  MoveL 1304 to (49.51, 43.02, 7) mm, rotated rx 0 ry 90 rz 0 deg; joints [-9.498, 3.635, 52.807, 168.647, 56.961, -173.753]
  Set speed (120.0 mm/s)
  MoveL 1305 to (57.59, 48.33, 7) mm, rotated rx 0 ry 90 rz 0 deg; joints [-9.745, 4.388, 50.732, 168.176, 55.695, -173.271]
  Set speed (1000.0 mm/s)
  MoveL 1306 to (57.66, 48.4, 7) mm, rotated rx 0 ry 90 rz 0 deg; joints [-9.748, 4.395, 50.713, 168.17, 55.683, -173.265]
  Set speed (30.0 mm/s)
  Call Extruder(793.550)
  MoveL 1307 to (57.66, 50.87, 7) mm, rotated rx 0 ry 90 rz 0 deg; joints [-9.903, 4.432, 50.611, 167.975, 55.638, -173.145]
  Call Extruder(793.809)
  MoveL 1308 to (59.6, 50.88, 7) mm, rotated rx 0 ry 90 rz 0 deg; joints [-9.882, 4.602, 50.15, 167.959, 55.35, -173.085]
  Call Extruder(794.969)
  MoveL 1309 to (59.6, 59.6, 7) mm, rotated rx 0 ry 90 rz 0 deg; joints [-10.423, 4.74, 49.776, 167.271, 55.187, -172.651]
  Call Extruder(797.524)
  MoveL 1310 to (40.4, 59.6, 7) mm, rotated rx 0 ry 90 rz 0 deg; joints [-10.646, 3.144, 54.181, 167.412, 57.955, -173.243]
  Call Extruder(800.078)
  MoveL 1311 to (40.4, 40.4, 7) mm, rotated rx 0 ry 90 rz 0 deg; joints [-9.429, 2.881, 54.923, 168.897, 58.29, -174.111]
  Call Extruder(800.872)
  MoveL 1312 to (46.37, 40.4, 7) mm, rotated rx 0 ry 90 rz 0 deg; joints [-9.366, 3.347, 53.61, 168.868, 57.452, -173.957]
  Call Extruder(801.125)
  MoveL 1313 to (46.37, 42.3, 7) mm, rotated rx 0 ry 90 rz 0 deg; joints [-9.486, 3.372, 53.539, 168.721, 57.42, -173.871]
  Call Extruder(801.408)
  MoveL 1314 to (48.5, 42.29, 7) mm, rotated rx 0 ry 90 rz 0 deg; joints [-9.463, 3.543, 53.062, 168.71, 57.118, -173.814]
  Call Extruder(801.461)
  MoveL 1315 to (48.9, 42.29, 7) mm, rotated rx 0 ry 90 rz 0 deg; joints [-9.459, 3.575, 52.972, 168.707, 57.06, -173.803]
  Call Extruder(801.495)
  MoveL 1316 to (48.9, 41.89, 7) mm, rotated rx 0 ry 90 rz 0 deg; joints [-9.434, 3.57, 52.987, 168.738, 57.067, -173.821]
  Call Extruder(801.694)
  MoveL 1317 to (48.9, 40.4, 7) mm, rotated rx 0 ry 90 rz 0 deg; joints [-9.34, 3.55, 53.043, 168.854, 57.092, -173.89]
  Call Extruder(801.871)
  MoveL 1318 to (50.23, 40.4, 7) mm, rotated rx 0 ry 90 rz 0 deg; joints [-9.326, 3.658, 52.742, 168.846, 56.901, -173.855]
  Call Extruder(802.070)
  MoveL 1319 to (50.23, 41.9, 7) mm, rotated rx 0 ry 90 rz 0 deg; joints [-9.42, 3.678, 52.686, 168.73, 56.876, -173.785]
  Call Extruder(802.124)
  MoveL 1320 to (50.23, 42.3, 7) mm, rotated rx 0 ry 90 rz 0 deg; joints [-9.445, 3.683, 52.671, 168.699, 56.87, -173.767]
  Call Extruder(802.158)
  MoveL 1321 to (50.63, 42.3, 7) mm, rotated rx 0 ry 90 rz 0 deg; joints [-9.441, 3.716, 52.58, 168.697, 56.812, -173.756]
  Call Extruder(802.438)
  MoveL 1322 to (52.74, 42.3, 7) mm, rotated rx 0 ry 90 rz 0 deg; joints [-9.419, 3.89, 52.098, 168.683, 56.508, -173.698]
  Call Extruder(802.691)
  MoveL 1323 to (52.74, 40.4, 7) mm, rotated rx 0 ry 90 rz 0 deg; joints [-9.3, 3.865, 52.169, 168.831, 56.54, -173.787]
  Call Extruder(803.603)
  MoveL 1324 to (59.6, 40.4, 7) mm, rotated rx 0 ry 90 rz 0 deg; joints [-9.23, 4.447, 50.57, 168.782, 55.535, -173.596]
  Call Extruder(804.666)
  MoveL 1325 to (59.6, 48.39, 7) mm, rotated rx 0 ry 90 rz 0 deg; joints [-9.728, 4.564, 50.252, 168.154, 55.395, -173.207]
  Call Extruder(804.925)
  MoveL 1326 to (57.66, 48.4, 7) mm, rotated rx 0 ry 90 rz 0 deg; joints [-9.748, 4.395, 50.713, 168.17, 55.683, -173.265]
  Set speed (120.0 mm/s)
  MoveL 1327 to (57.66, 48.8, 7) mm, rotated rx 0 ry 90 rz 0 deg; joints [-9.773, 4.401, 50.697, 168.139, 55.676, -173.246]
  Set speed (1000.0 mm/s)
  MoveL 1328 to (57.56, 48.8, 7) mm, rotated rx 0 ry 90 rz 0 deg; joints [-9.774, 4.392, 50.72, 168.139, 55.691, -173.249]
  MoveL 1329 to (49.86, 42.5, 7) mm, rotated rx 0 ry 90 rz 0 deg; joints [-9.462, 3.656, 52.748, 168.685, 56.92, -173.767]
  MoveL 1330 to (49.57, 42.21, 7) mm, rotated rx 0 ry 90 rz 0 deg; joints [-9.447, 3.628, 52.825, 168.71, 56.967, -173.789]
  Set speed (30.0 mm/s)
  Call Extruder(804.972)
  MoveL 1331 to (49.57, 41.65, 7) mm, rotated rx 0 ry 90 rz 0 deg; joints [-9.411, 3.62, 52.846, 168.754, 56.976, -173.815]
  Call Extruder(805.055)
  MoveL 1332 to (49.4, 42.61, 7) mm, rotated rx 0 ry 90 rz 0 deg; joints [-9.474, 3.62, 52.848, 168.68, 56.984, -173.775]
  Set speed (120.0 mm/s)
  MoveL 1333 to (49.47, 42.86, 7) mm, rotated rx 0 ry 90 rz 0 deg; joints [-9.489, 3.629, 52.823, 168.66, 56.97, -173.762]
  Set speed (1000.0 mm/s)
  MoveL 1334 to (49.27, 43.01, 7) mm, rotated rx 0 ry 90 rz 0 deg; joints [-9.501, 3.615, 52.862, 168.649, 56.996, -173.76]
  MoveL 1335 to (49.27, 43.01, 7.4) mm, rotated rx 0 ry 90 rz 0 deg; joints [-9.501, 3.572, 52.909, 168.65, 56.999, -173.761]
  Set speed (60.0 mm/s)
  Call Extruder(805.506)
  MoveL 1336 to (45.88, 43.01, 7.4) mm, rotated rx 0 ry 90 rz 0 deg; joints [-9.537, 3.299, 53.669, 168.669, 57.482, -173.852]
  Call Extruder(805.533)
  MoveL 1337 to (45.88, 42.81, 7.4) mm, rotated rx 0 ry 90 rz 0 deg; joints [-9.524, 3.296, 53.677, 168.685, 57.486, -173.861]
  Call Extruder(806.428)
  MoveL 1338 to (41.12, 47.56, 7.4) mm, rotated rx 0 ry 90 rz 0 deg; joints [-9.876, 2.988, 54.547, 168.341, 58.073, -173.772]
  Call Extruder(807.286)
  MoveL 1339 to (41.12, 41.12, 7.4) mm, rotated rx 0 ry 90 rz 0 deg; joints [-9.467, 2.903, 54.786, 168.839, 58.181, -174.061]
  Call Extruder(810.627)
  MoveL 1340 to (58.88, 58.88, 7.4) mm, rotated rx 0 ry 90 rz 0 deg; joints [-10.386, 4.621, 50.029, 167.335, 55.313, -172.712]
  Call Extruder(810.627)
  MoveL 1341 to (58.88, 58.88, 7.4) mm, rotated rx 0 ry 90 rz 0 deg; joints [-10.386, 4.621, 50.029, 167.335, 55.313, -172.712]
  Call Extruder(811.485)
  MoveL 1342 to (58.88, 52.43, 7.4) mm, rotated rx 0 ry 90 rz 0 deg; joints [-9.986, 4.519, 50.306, 167.843, 55.434, -173.032]
  Call Extruder(812.698)
  MoveL 1343 to (52.43, 58.88, 7.4) mm, rotated rx 0 ry 90 rz 0 deg; joints [-10.46, 4.064, 51.546, 167.39, 56.26, -172.917]
  Call Extruder(813.345)
  MoveL 1344 to (47.57, 58.88, 7.4) mm, rotated rx 0 ry 90 rz 0 deg; joints [-10.516, 3.661, 52.661, 167.425, 56.961, -173.066]
  Call Extruder(814.558)
  MoveL 1345 to (41.12, 52.43, 7.4) mm, rotated rx 0 ry 90 rz 0 deg; joints [-10.184, 3.054, 54.358, 167.964, 57.988, -173.552]
  Call Extruder(815.416)
  MoveL 1346 to (41.12, 58.88, 7.4) mm, rotated rx 0 ry 90 rz 0 deg; joints [-10.592, 3.146, 54.099, 167.464, 57.871, -173.256]
  Call Extruder(815.416)
  MoveL 1347 to (41.12, 58.88, 7.4) mm, rotated rx 0 ry 90 rz 0 deg; joints [-10.592, 3.146, 54.099, 167.464, 57.871, -173.256]
  Call Extruder(818.758)
  MoveL 1348 to (58.88, 41.12, 7.4) mm, rotated rx 0 ry 90 rz 0 deg; joints [-9.282, 4.351, 50.761, 168.732, 55.634, -173.583]
  Call Extruder(819.615)
  MoveL 1349 to (58.88, 47.56, 7.4) mm, rotated rx 0 ry 90 rz 0 deg; joints [-9.684, 4.445, 50.506, 168.226, 55.522, -173.27]
  Call Extruder(820.682)
  MoveL 1350 to (53.21, 41.89, 7.4) mm, rotated rx 0 ry 90 rz 0 deg; joints [-9.389, 3.88, 52.054, 168.712, 56.451, -173.705]
  MoveL 1351 to (53.07, 41.75, 7.4) mm, rotated rx 0 ry 90 rz 0 deg; joints [-9.382, 3.866, 52.092, 168.724, 56.474, -173.716]
  Set speed (120.0 mm/s)
  MoveL 1352 to (49.27, 43.02, 7.4) mm, rotated rx 0 ry 90 rz 0 deg; joints [-9.501, 3.572, 52.909, 168.649, 56.999, -173.761]
  Set speed (60.0 mm/s)
  Call Extruder(821.206)
  MoveL 1353 to (53.21, 43.02, 7.4) mm, rotated rx 0 ry 90 rz 0 deg; joints [-9.459, 3.896, 52.011, 168.624, 56.432, -173.652]
  Call Extruder(821.458)
  MoveL 1354 to (53.21, 41.12, 7.4) mm, rotated rx 0 ry 90 rz 0 deg; joints [-9.34, 3.87, 52.082, 168.772, 56.464, -173.741]
  Call Extruder(822.213)
  MoveL 1355 to (58.88, 41.12, 7.4) mm, rotated rx 0 ry 90 rz 0 deg; joints [-9.282, 4.351, 50.761, 168.731, 55.634, -173.583]
  MoveL 1356 to (59.08, 41.12, 7.4) mm, rotated rx 0 ry 90 rz 0 deg; joints [-9.28, 4.369, 50.714, 168.73, 55.604, -173.577]
  Set speed (120.0 mm/s)
  MoveL 1357 to (49.27, 43.01, 7.4) mm, rotated rx 0 ry 90 rz 0 deg; joints [-9.501, 3.572, 52.909, 168.65, 56.999, -173.761]
  Set speed (60.0 mm/s)
  Call Extruder(822.213)
  MoveL 1358 to (49.27, 43.02, 7.4) mm, rotated rx 0 ry 90 rz 0 deg; joints [-9.501, 3.572, 52.909, 168.649, 56.999, -173.761]
  Set speed (120.0 mm/s)
  MoveL 1359 to (57.59, 48.32, 7.4) mm, rotated rx 0 ry 90 rz 0 deg; joints [-9.745, 4.344, 50.781, 168.177, 55.699, -173.272]
  Set speed (1000.0 mm/s)
  MoveL 1360 to (57.66, 48.39, 7.4) mm, rotated rx 0 ry 90 rz 0 deg; joints [-9.748, 4.351, 50.761, 168.171, 55.687, -173.267]
  Set speed (30.0 mm/s)
  Call Extruder(822.543)
  MoveL 1361 to (57.66, 50.87, 7.4) mm, rotated rx 0 ry 90 rz 0 deg; joints [-9.903, 4.388, 50.66, 167.976, 55.643, -173.146]
  Call Extruder(822.801)
  MoveL 1362 to (59.6, 50.87, 7.4) mm, rotated rx 0 ry 90 rz 0 deg; joints [-9.882, 4.558, 50.199, 167.96, 55.355, -173.086]
  Call Extruder(823.962)
  MoveL 1363 to (59.6, 59.6, 7.4) mm, rotated rx 0 ry 90 rz 0 deg; joints [-10.423, 4.696, 49.825, 167.271, 55.192, -172.653]
  Call Extruder(826.517)
  MoveL 1364 to (40.4, 59.6, 7.4) mm, rotated rx 0 ry 90 rz 0 deg; joints [-10.646, 3.101, 54.227, 167.412, 57.958, -173.244]
  Call Extruder(829.071)
  MoveL 1365 to (40.4, 40.4, 7.4) mm, rotated rx 0 ry 90 rz 0 deg; joints [-9.429, 2.839, 54.968, 168.898, 58.293, -174.112]
  Call Extruder(829.895)
  MoveL 1366 to (46.59, 40.4, 7.4) mm, rotated rx 0 ry 90 rz 0 deg; joints [-9.364, 3.322, 53.607, 168.868, 57.424, -173.952]
  Call Extruder(830.147)
  MoveL 1367 to (46.6, 42.29, 7.4) mm, rotated rx 0 ry 90 rz 0 deg; joints [-9.483, 3.347, 53.536, 168.721, 57.392, -173.866]
  Call Extruder(830.432)
  MoveL 1368 to (48.74, 42.29, 7.4) mm, rotated rx 0 ry 90 rz 0 deg; joints [-9.461, 3.519, 53.056, 168.709, 57.087, -173.808]
  Call Extruder(830.485)
  MoveL 1369 to (49.14, 42.29, 7.4) mm, rotated rx 0 ry 90 rz 0 deg; joints [-9.457, 3.551, 52.965, 168.706, 57.03, -173.797]
  Call Extruder(830.520)
  MoveL 1370 to (49.14, 41.89, 7.4) mm, rotated rx 0 ry 90 rz 0 deg; joints [-9.431, 3.546, 52.98, 168.737, 57.037, -173.816]
  Call Extruder(830.719)
  MoveL 1371 to (49.14, 40.4, 7.4) mm, rotated rx 0 ry 90 rz 0 deg; joints [-9.337, 3.526, 53.036, 168.853, 57.062, -173.885]
  Call Extruder(830.832)
  MoveL 1372 to (49.99, 40.4, 7.4) mm, rotated rx 0 ry 90 rz 0 deg; joints [-9.328, 3.595, 52.844, 168.848, 56.94, -173.862]
  Call Extruder(831.031)
  MoveL 1373 to (49.99, 41.9, 7.4) mm, rotated rx 0 ry 90 rz 0 deg; joints [-9.423, 3.615, 52.788, 168.732, 56.915, -173.793]
  Call Extruder(831.084)
  MoveL 1374 to (49.99, 42.29, 7.4) mm, rotated rx 0 ry 90 rz 0 deg; joints [-9.448, 3.62, 52.773, 168.701, 56.908, -173.774]
  Call Extruder(831.118)
  MoveL 1375 to (50.39, 42.3, 7.4) mm, rotated rx 0 ry 90 rz 0 deg; joints [-9.444, 3.653, 52.682, 168.699, 56.851, -173.764]
  Call Extruder(831.398)
  MoveL 1376 to (52.49, 42.3, 7.4) mm, rotated rx 0 ry 90 rz 0 deg; joints [-9.422, 3.826, 52.204, 168.685, 56.549, -173.706]
  Call Extruder(831.650)
  MoveL 1377 to (52.49, 40.4, 7.4) mm, rotated rx 0 ry 90 rz 0 deg; joints [-9.303, 3.8, 52.274, 168.833, 56.58, -173.795]
  Call Extruder(832.596)
  MoveL 1378 to (59.6, 40.4, 7.4) mm, rotated rx 0 ry 90 rz 0 deg; joints [-9.23, 4.404, 50.618, 168.782, 55.539, -173.597]
  Call Extruder(833.659)
  MoveL 1379 to (59.6, 48.39, 7.4) mm, rotated rx 0 ry 90 rz 0 deg; joints [-9.727, 4.52, 50.301, 168.155, 55.4, -173.208]
  Call Extruder(833.917)
  MoveL 1380 to (57.66, 48.39, 7.4) mm, rotated rx 0 ry 90 rz 0 deg; joints [-9.748, 4.351, 50.761, 168.171, 55.687, -173.267]
  Set speed (120.0 mm/s)
  MoveL 1381 to (57.66, 48.79, 7.4) mm, rotated rx 0 ry 90 rz 0 deg; joints [-9.773, 4.357, 50.745, 168.14, 55.68, -173.247]
  Set speed (1000.0 mm/s)
  MoveL 1382 to (57.56, 48.79, 7.4) mm, rotated rx 0 ry 90 rz 0 deg; joints [-9.774, 4.349, 50.769, 168.14, 55.695, -173.25]
  MoveL 1383 to (49.61, 42.59, 7.4) mm, rotated rx 0 ry 90 rz 0 deg; joints [-9.47, 3.594, 52.847, 168.68, 56.957, -173.771]
  MoveL 1384 to (49.56, 42.64, 7.4) mm, rotated rx 0 ry 90 rz 0 deg; joints [-9.474, 3.59, 52.857, 168.677, 56.964, -173.77]
  Set speed (30.0 mm/s)
  Call Extruder(833.929)
  MoveL 1385 to (49.56, 42.08, 7.4) mm, rotated rx 0 ry 90 rz 0 deg; joints [-9.439, 3.583, 52.878, 168.721, 56.973, -173.796]
  Call Extruder(833.954)
  MoveL 1386 to (49.56, 40.95, 7.4) mm, rotated rx 0 ry 90 rz 0 deg; joints [-9.367, 3.568, 52.92, 168.808, 56.992, -173.848]
  Set speed (120.0 mm/s)
  MoveL 1387 to (49.94, 40.9, 7.4) mm, rotated rx 0 ry 90 rz 0 deg; joints [-9.36, 3.597, 52.837, 168.81, 56.939, -173.841]
  Set speed (1000.0 mm/s)
  MoveL 1388 to (49.89, 40.9, 7.4) mm, rotated rx 0 ry 90 rz 0 deg; joints [-9.361, 3.594, 52.848, 168.81, 56.946, -173.842]
  MoveL 1389 to (49.02, 43.01, 7.4) mm, rotated rx 0 ry 90 rz 0 deg; joints [-9.503, 3.552, 52.964, 168.651, 57.035, -173.767]
  MoveL 1390 to (49.02, 43.01, 7.8) mm, rotated rx 0 ry 90 rz 0 deg; joints [-9.503, 3.509, 53.011, 168.651, 57.038, -173.768]
  Set speed (60.0 mm/s)
  Call Extruder(834.343)
  MoveL 1391 to (46.1, 43.02, 7.8) mm, rotated rx 0 ry 90 rz 0 deg; joints [-9.534, 3.274, 53.666, 168.668, 57.454, -173.847]
  Call Extruder(834.400)
  MoveL 1392 to (46.1, 42.59, 7.8) mm, rotated rx 0 ry 90 rz 0 deg; joints [-9.507, 3.268, 53.682, 168.701, 57.461, -173.866]
  Call Extruder(835.337)
  MoveL 1393 to (41.12, 47.56, 7.8) mm, rotated rx 0 ry 90 rz 0 deg; joints [-9.876, 2.945, 54.592, 168.341, 58.076, -173.773]
  Call Extruder(836.194)
  MoveL 1394 to (41.12, 41.12, 7.8) mm, rotated rx 0 ry 90 rz 0 deg; joints [-9.467, 2.86, 54.832, 168.839, 58.184, -174.062]
  Call Extruder(839.536)
  MoveL 1395 to (58.88, 58.88, 7.8) mm, rotated rx 0 ry 90 rz 0 deg; joints [-10.386, 4.577, 50.078, 167.336, 55.318, -172.714]
  Call Extruder(839.536)
  MoveL 1396 to (58.88, 58.88, 7.8) mm, rotated rx 0 ry 90 rz 0 deg; joints [-10.386, 4.577, 50.078, 167.336, 55.318, -172.714]
  Call Extruder(840.394)
  MoveL 1397 to (58.88, 52.43, 7.8) mm, rotated rx 0 ry 90 rz 0 deg; joints [-9.986, 4.475, 50.354, 167.844, 55.439, -173.033]
  Call Extruder(841.606)
  MoveL 1398 to (52.43, 58.88, 7.8) mm, rotated rx 0 ry 90 rz 0 deg; joints [-10.46, 4.021, 51.594, 167.39, 56.264, -172.918]
  Call Extruder(842.254)
  MoveL 1399 to (47.56, 58.88, 7.8) mm, rotated rx 0 ry 90 rz 0 deg; joints [-10.516, 3.618, 52.708, 167.425, 56.964, -173.067]
  Call Extruder(843.467)
  MoveL 1400 to (41.12, 52.43, 7.8) mm, rotated rx 0 ry 90 rz 0 deg; joints [-10.184, 3.012, 54.404, 167.964, 57.991, -173.552]
  Call Extruder(844.324)
  MoveL 1401 to (41.12, 58.88, 7.8) mm, rotated rx 0 ry 90 rz 0 deg; joints [-10.592, 3.104, 54.145, 167.464, 57.874, -173.257]
  Call Extruder(844.325)
  MoveL 1402 to (41.12, 58.88, 7.8) mm, rotated rx 0 ry 90 rz 0 deg; joints [-10.592, 3.104, 54.145, 167.464, 57.874, -173.257]
  Call Extruder(847.666)
  MoveL 1403 to (58.88, 41.12, 7.8) mm, rotated rx 0 ry 90 rz 0 deg; joints [-9.282, 4.308, 50.81, 168.732, 55.639, -173.584]
  Call Extruder(848.524)
  MoveL 1404 to (58.88, 47.56, 7.8) mm, rotated rx 0 ry 90 rz 0 deg; joints [-9.684, 4.401, 50.555, 168.227, 55.527, -173.272]
  Call Extruder(849.638)
  MoveL 1405 to (52.96, 41.64, 7.8) mm, rotated rx 0 ry 90 rz 0 deg; joints [-9.376, 3.812, 52.168, 168.734, 56.496, -173.725]
  MoveL 1406 to (52.81, 41.5, 7.8) mm, rotated rx 0 ry 90 rz 0 deg; joints [-9.368, 3.799, 52.206, 168.746, 56.519, -173.735]
  Set speed (120.0 mm/s)
  MoveL 1407 to (49.02, 43.02, 7.8) mm, rotated rx 0 ry 90 rz 0 deg; joints [-9.503, 3.509, 53.011, 168.651, 57.038, -173.768]
  Set speed (60.0 mm/s)
  Call Extruder(850.161)
  MoveL 1408 to (52.95, 43.02, 7.8) mm, rotated rx 0 ry 90 rz 0 deg; joints [-9.462, 3.831, 52.116, 168.626, 56.473, -173.66]
  Call Extruder(850.414)
  MoveL 1409 to (52.96, 41.12, 7.8) mm, rotated rx 0 ry 90 rz 0 deg; joints [-9.343, 3.805, 52.188, 168.774, 56.504, -173.749]
  Call Extruder(851.202)
  MoveL 1410 to (58.88, 41.12, 7.8) mm, rotated rx 0 ry 90 rz 0 deg; joints [-9.282, 4.308, 50.809, 168.732, 55.638, -173.584]
  MoveL 1411 to (59.08, 41.12, 7.8) mm, rotated rx 0 ry 90 rz 0 deg; joints [-9.28, 4.325, 50.762, 168.731, 55.609, -173.578]
  Set speed (120.0 mm/s)
  MoveL 1412 to (49.02, 43.01, 7.8) mm, rotated rx 0 ry 90 rz 0 deg; joints [-9.503, 3.509, 53.011, 168.651, 57.038, -173.768]
  Set speed (60.0 mm/s)
  Call Extruder(851.202)
  MoveL 1413 to (49.02, 43.02, 7.8) mm, rotated rx 0 ry 90 rz 0 deg; joints [-9.503, 3.509, 53.011, 168.651, 57.038, -173.768]
  Set speed (120.0 mm/s)
  MoveL 1414 to (49.74, 42.29, 7.8) mm, rotated rx 0 ry 90 rz 0 deg; joints [-9.45, 3.557, 52.875, 168.703, 56.947, -173.782]
  Set speed (30.0 mm/s)
  Call Extruder(851.533)
  MoveL 1415 to (52.24, 42.3, 7.8) mm, rotated rx 0 ry 90 rz 0 deg; joints [-9.424, 3.762, 52.309, 168.687, 56.589, -173.714]
  Call Extruder(851.785)
  MoveL 1416 to (52.24, 40.4, 7.8) mm, rotated rx 0 ry 90 rz 0 deg; joints [-9.305, 3.736, 52.379, 168.835, 56.62, -173.803]
  Call Extruder(852.765)
  MoveL 1417 to (59.6, 40.4, 7.8) mm, rotated rx 0 ry 90 rz 0 deg; joints [-9.23, 4.36, 50.667, 168.783, 55.544, -173.598]
  Call Extruder(853.827)
  MoveL 1418 to (59.6, 48.39, 7.8) mm, rotated rx 0 ry 90 rz 0 deg; joints [-9.727, 4.476, 50.35, 168.156, 55.405, -173.21]
  Call Extruder(854.032)
  MoveL 1419 to (58.06, 48.39, 7.8) mm, rotated rx 0 ry 90 rz 0 deg; joints [-9.744, 4.342, 50.715, 168.169, 55.633, -173.256]
  Call Extruder(854.085)
  MoveL 1420 to (57.66, 48.39, 7.8) mm, rotated rx 0 ry 90 rz 0 deg; joints [-9.748, 4.308, 50.81, 168.172, 55.692, -173.268]
  Call Extruder(854.120)
  MoveL 1421 to (57.66, 48.79, 7.8) mm, rotated rx 0 ry 90 rz 0 deg; joints [-9.773, 4.314, 50.793, 168.141, 55.685, -173.249]
  Call Extruder(854.396)
  MoveL 1422 to (57.66, 50.87, 7.8) mm, rotated rx 0 ry 90 rz 0 deg; joints [-9.902, 4.345, 50.708, 167.977, 55.647, -173.147]
  Call Extruder(854.654)
  MoveL 1423 to (59.6, 50.87, 7.8) mm, rotated rx 0 ry 90 rz 0 deg; joints [-9.881, 4.514, 50.248, 167.961, 55.36, -173.088]
  Call Extruder(855.816)
  MoveL 1424 to (59.6, 59.6, 7.8) mm, rotated rx 0 ry 90 rz 0 deg; joints [-10.423, 4.652, 49.874, 167.272, 55.197, -172.654]
  Call Extruder(858.370)
  MoveL 1425 to (40.4, 59.6, 7.8) mm, rotated rx 0 ry 90 rz 0 deg; joints [-10.646, 3.058, 54.273, 167.412, 57.961, -173.244]
  Call Extruder(860.925)
  MoveL 1426 to (40.4, 40.4, 7.8) mm, rotated rx 0 ry 90 rz 0 deg; joints [-9.429, 2.796, 55.014, 168.898, 58.296, -174.112]
  Call Extruder(861.778)
  MoveL 1427 to (46.82, 40.4, 7.8) mm, rotated rx 0 ry 90 rz 0 deg; joints [-9.361, 3.297, 53.603, 168.867, 57.396, -173.947]
  Call Extruder(862.030)
  MoveL 1428 to (46.82, 42.3, 7.8) mm, rotated rx 0 ry 90 rz 0 deg; joints [-9.481, 3.322, 53.533, 168.72, 57.364, -173.86]
  Call Extruder(862.371)
  MoveL 1429 to (49.37, 42.29, 7.8) mm, rotated rx 0 ry 90 rz 0 deg; joints [-9.454, 3.527, 52.959, 168.705, 57, -173.792]
  Call Extruder(862.474)
  MoveL 1430 to (49.37, 41.52, 7.8) mm, rotated rx 0 ry 90 rz 0 deg; joints [-9.405, 3.517, 52.988, 168.766, 57.013, -173.828]
  Call Extruder(862.623)
  MoveL 1431 to (49.37, 40.4, 7.8) mm, rotated rx 0 ry 90 rz 0 deg; joints [-9.335, 3.502, 53.029, 168.852, 57.032, -173.879]
  Call Extruder(862.672)
  MoveL 1432 to (49.75, 40.4, 7.8) mm, rotated rx 0 ry 90 rz 0 deg; joints [-9.331, 3.532, 52.945, 168.85, 56.978, -173.87]
  Call Extruder(862.741)
  MoveL 1433 to (49.75, 41.52, 7.8) mm, rotated rx 0 ry 90 rz 0 deg; joints [-9.401, 3.547, 52.904, 168.764, 56.96, -173.818]
  Call Extruder(862.789)
  MoveL 1434 to (49.74, 42.29, 7.8) mm, rotated rx 0 ry 90 rz 0 deg; joints [-9.45, 3.557, 52.875, 168.703, 56.947, -173.782]
  Set speed (120.0 mm/s)
  MoveL 1435 to (50.14, 42.29, 7.8) mm, rotated rx 0 ry 90 rz 0 deg; joints [-9.446, 3.59, 52.785, 168.701, 56.89, -173.771]
  Set speed (1000.0 mm/s)
  MoveL 1436 to (50.14, 43.1, 7.8) mm, rotated rx 0 ry 90 rz 0 deg; joints [-9.496, 3.601, 52.754, 168.638, 56.876, -173.734]
  MoveL 1437 to (52.26, 42.32, 7.8) mm, rotated rx 0 ry 90 rz 0 deg; joints [-9.426, 3.764, 52.301, 168.685, 56.585, -173.712]
  MoveL 1438 to (52.7, 41.39, 7.8) mm, rotated rx 0 ry 90 rz 0 deg; joints [-9.363, 3.788, 52.236, 168.755, 56.537, -173.744]
  MoveL 1439 to (52.7, 41.39, 8.2) mm, rotated rx 0 ry 90 rz 0 deg; joints [-9.363, 3.745, 52.283, 168.755, 56.541, -173.745]
  Set speed (60.0 mm/s)
  Call Extruder(863.951)
  MoveL 1440 to (58.88, 47.57, 8.2) mm, rotated rx 0 ry 90 rz 0 deg; joints [-9.684, 4.357, 50.603, 168.227, 55.531, -173.273]
  Call Extruder(864.809)
  MoveL 1441 to (58.88, 41.12, 8.2) mm, rotated rx 0 ry 90 rz 0 deg; joints [-9.282, 4.264, 50.858, 168.733, 55.643, -173.585]
  Call Extruder(868.150)
  MoveL 1442 to (41.12, 58.88, 8.2) mm, rotated rx 0 ry 90 rz 0 deg; joints [-10.592, 3.061, 54.191, 167.465, 57.877, -173.258]
  Call Extruder(868.151)
  MoveL 1443 to (41.12, 58.88, 8.2) mm, rotated rx 0 ry 90 rz 0 deg; joints [-10.592, 3.061, 54.19, 167.465, 57.877, -173.257]
  Call Extruder(869.008)
  MoveL 1444 to (41.12, 52.43, 8.2) mm, rotated rx 0 ry 90 rz 0 deg; joints [-10.184, 2.969, 54.45, 167.965, 57.994, -173.553]
  Call Extruder(870.221)
  MoveL 1445 to (47.57, 58.88, 8.2) mm, rotated rx 0 ry 90 rz 0 deg; joints [-10.516, 3.575, 52.755, 167.426, 56.968, -173.068]
  Call Extruder(870.869)
  MoveL 1446 to (52.43, 58.88, 8.2) mm, rotated rx 0 ry 90 rz 0 deg; joints [-10.46, 3.978, 51.642, 167.391, 56.268, -172.919]
  Call Extruder(872.082)
  MoveL 1447 to (58.88, 52.43, 8.2) mm, rotated rx 0 ry 90 rz 0 deg; joints [-9.986, 4.431, 50.403, 167.844, 55.443, -173.034]
  Call Extruder(872.939)
  MoveL 1448 to (58.88, 58.88, 8.2) mm, rotated rx 0 ry 90 rz 0 deg; joints [-10.386, 4.533, 50.127, 167.336, 55.323, -172.715]
  Call Extruder(872.940)
  MoveL 1449 to (58.88, 58.88, 8.2) mm, rotated rx 0 ry 90 rz 0 deg; joints [-10.386, 4.533, 50.127, 167.337, 55.323, -172.715]
  Call Extruder(876.281)
  MoveL 1450 to (41.12, 41.12, 8.2) mm, rotated rx 0 ry 90 rz 0 deg; joints [-9.467, 2.818, 54.877, 168.84, 58.187, -174.063]
  Call Extruder(877.139)
  MoveL 1451 to (41.12, 47.56, 8.2) mm, rotated rx 0 ry 90 rz 0 deg; joints [-9.876, 2.902, 54.638, 168.342, 58.079, -173.774]
  Call Extruder(878.117)
  MoveL 1452 to (46.32, 42.37, 8.2) mm, rotated rx 0 ry 90 rz 0 deg; joints [-9.491, 3.24, 53.687, 168.718, 57.437, -173.871]
  Call Extruder(878.203)
  MoveL 1453 to (46.32, 43.02, 8.2) mm, rotated rx 0 ry 90 rz 0 deg; joints [-9.532, 3.249, 53.663, 168.667, 57.426, -173.841]
  Call Extruder(879.052)
  MoveL 1454 to (52.7, 43.02, 8.2) mm, rotated rx 0 ry 90 rz 0 deg; joints [-9.465, 3.767, 52.222, 168.629, 56.513, -173.668]
  Call Extruder(879.304)
  MoveL 1455 to (52.7, 41.12, 8.2) mm, rotated rx 0 ry 90 rz 0 deg; joints [-9.346, 3.741, 52.293, 168.776, 56.545, -173.757]
  Call Extruder(880.126)
  MoveL 1456 to (58.88, 41.12, 8.2) mm, rotated rx 0 ry 90 rz 0 deg; joints [-9.282, 4.264, 50.858, 168.733, 55.643, -173.585]
  MoveL 1457 to (59.08, 41.12, 8.2) mm, rotated rx 0 ry 90 rz 0 deg; joints [-9.28, 4.281, 50.81, 168.731, 55.613, -173.579]
  Set speed (120.0 mm/s)
  MoveL 1458 to (57.59, 48.31, 8.2) mm, rotated rx 0 ry 90 rz 0 deg; joints [-9.744, 4.257, 50.877, 168.179, 55.708, -173.275]
  Set speed (1000.0 mm/s)
  MoveL 1459 to (57.66, 48.38, 8.2) mm, rotated rx 0 ry 90 rz 0 deg; joints [-9.748, 4.264, 50.858, 168.173, 55.696, -173.269]
  Set speed (30.0 mm/s)
  Call Extruder(880.353)
  MoveL 1460 to (57.66, 50.09, 8.2) mm, rotated rx 0 ry 90 rz 0 deg; joints [-9.854, 4.289, 50.789, 168.039, 55.666, -173.186]
  Call Extruder(880.456)
  MoveL 1461 to (57.66, 50.86, 8.2) mm, rotated rx 0 ry 90 rz 0 deg; joints [-9.902, 4.301, 50.756, 167.978, 55.652, -173.149]
  Call Extruder(880.714)
  MoveL 1462 to (59.6, 50.86, 8.2) mm, rotated rx 0 ry 90 rz 0 deg; joints [-9.881, 4.47, 50.297, 167.962, 55.365, -173.089]
  Call Extruder(881.876)
  MoveL 1463 to (59.6, 59.6, 8.2) mm, rotated rx 0 ry 90 rz 0 deg; joints [-10.423, 4.608, 49.923, 167.273, 55.202, -172.655]
  Call Extruder(884.430)
  MoveL 1464 to (40.4, 59.6, 8.2) mm, rotated rx 0 ry 90 rz 0 deg; joints [-10.646, 3.015, 54.319, 167.413, 57.964, -173.245]
  Call Extruder(886.985)
  MoveL 1465 to (40.4, 40.4, 8.2) mm, rotated rx 0 ry 90 rz 0 deg; joints [-9.429, 2.754, 55.059, 168.898, 58.299, -174.113]
  Call Extruder(887.868)
  MoveL 1466 to (47.04, 40.4, 8.2) mm, rotated rx 0 ry 90 rz 0 deg; joints [-9.359, 3.271, 53.6, 168.866, 57.368, -173.942]
  Call Extruder(888.120)
  MoveL 1467 to (47.04, 42.3, 8.2) mm, rotated rx 0 ry 90 rz 0 deg; joints [-9.479, 3.297, 53.529, 168.719, 57.336, -173.855]
  Call Extruder(888.778)
  MoveL 1468 to (51.98, 42.3, 8.2) mm, rotated rx 0 ry 90 rz 0 deg; joints [-9.427, 3.698, 52.413, 168.689, 56.629, -173.722]
  Call Extruder(889.030)
  MoveL 1469 to (51.99, 40.4, 8.2) mm, rotated rx 0 ry 90 rz 0 deg; joints [-9.308, 3.672, 52.484, 168.837, 56.661, -173.81]
  Call Extruder(890.043)
  MoveL 1470 to (59.6, 40.4, 8.2) mm, rotated rx 0 ry 90 rz 0 deg; joints [-9.23, 4.316, 50.715, 168.784, 55.549, -173.599]
  Call Extruder(891.105)
  MoveL 1471 to (59.6, 48.38, 8.2) mm, rotated rx 0 ry 90 rz 0 deg; joints [-9.727, 4.433, 50.399, 168.157, 55.41, -173.211]
  Call Extruder(891.363)
  MoveL 1472 to (57.66, 48.38, 8.2) mm, rotated rx 0 ry 90 rz 0 deg; joints [-9.748, 4.264, 50.858, 168.173, 55.696, -173.269]
  Set speed (120.0 mm/s)
  MoveL 1473 to (57.66, 48.78, 8.2) mm, rotated rx 0 ry 90 rz 0 deg; joints [-9.773, 4.27, 50.842, 168.142, 55.689, -173.25]
  Set speed (1000.0 mm/s)
  MoveL 1474 to (56.86, 48.78, 8.2) mm, rotated rx 0 ry 90 rz 0 deg; joints [-9.781, 4.201, 51.03, 168.148, 55.807, -173.274]
  MoveL 1475 to (52.45, 41.14, 8.2) mm, rotated rx 0 ry 90 rz 0 deg; joints [-9.349, 3.72, 52.351, 168.777, 56.581, -173.763]
  MoveL 1476 to (52.45, 41.14, 8.6) mm, rotated rx 0 ry 90 rz 0 deg; joints [-9.349, 3.677, 52.398, 168.777, 56.585, -173.764]
  Set speed (60.0 mm/s)
  Call Extruder(892.573)
  MoveL 1477 to (58.88, 47.57, 8.6) mm, rotated rx 0 ry 90 rz 0 deg; joints [-9.684, 4.314, 50.652, 168.228, 55.536, -173.274]
  Call Extruder(893.430)
  MoveL 1478 to (58.88, 41.12, 8.6) mm, rotated rx 0 ry 90 rz 0 deg; joints [-9.282, 4.22, 50.906, 168.733, 55.647, -173.586]
  Call Extruder(896.772)
  MoveL 1479 to (41.12, 58.88, 8.6) mm, rotated rx 0 ry 90 rz 0 deg; joints [-10.592, 3.018, 54.236, 167.465, 57.88, -173.258]
  Call Extruder(896.772)
  MoveL 1480 to (41.12, 58.88, 8.6) mm, rotated rx 0 ry 90 rz 0 deg; joints [-10.592, 3.018, 54.236, 167.465, 57.88, -173.258]
  Call Extruder(897.630)
  MoveL 1481 to (41.12, 52.43, 8.6) mm, rotated rx 0 ry 90 rz 0 deg; joints [-10.184, 2.926, 54.495, 167.965, 57.997, -173.554]
  Call Extruder(898.842)
  MoveL 1482 to (47.57, 58.88, 8.6) mm, rotated rx 0 ry 90 rz 0 deg; joints [-10.516, 3.532, 52.801, 167.426, 56.972, -173.068]
  Call Extruder(899.490)
  MoveL 1483 to (52.43, 58.88, 8.6) mm, rotated rx 0 ry 90 rz 0 deg; joints [-10.46, 3.934, 51.689, 167.391, 56.272, -172.92]
  Call Extruder(900.703)
  MoveL 1484 to (58.88, 52.43, 8.6) mm, rotated rx 0 ry 90 rz 0 deg; joints [-9.986, 4.387, 50.451, 167.845, 55.448, -173.036]
  Call Extruder(901.561)
  MoveL 1485 to (58.88, 58.88, 8.6) mm, rotated rx 0 ry 90 rz 0 deg; joints [-10.386, 4.489, 50.175, 167.337, 55.327, -172.716]
  Call Extruder(901.561)
  MoveL 1486 to (58.88, 58.88, 8.6) mm, rotated rx 0 ry 90 rz 0 deg; joints [-10.386, 4.489, 50.176, 167.337, 55.327, -172.716]
  Call Extruder(904.902)
  MoveL 1487 to (41.12, 41.12, 8.6) mm, rotated rx 0 ry 90 rz 0 deg; joints [-9.467, 2.775, 54.922, 168.84, 58.19, -174.063]
  Call Extruder(905.760)
  MoveL 1488 to (41.12, 47.56, 8.6) mm, rotated rx 0 ry 90 rz 0 deg; joints [-9.876, 2.86, 54.683, 168.342, 58.081, -173.774]
  Call Extruder(906.780)
  MoveL 1489 to (46.54, 42.14, 8.6) mm, rotated rx 0 ry 90 rz 0 deg; joints [-9.474, 3.212, 53.692, 168.734, 57.412, -173.876]
  Call Extruder(906.896)
  MoveL 1490 to (46.54, 43.02, 8.6) mm, rotated rx 0 ry 90 rz 0 deg; joints [-9.53, 3.224, 53.659, 168.666, 57.397, -173.836]
  Call Extruder(907.681)
  MoveL 1491 to (52.45, 43.02, 8.6) mm, rotated rx 0 ry 90 rz 0 deg; joints [-9.467, 3.703, 52.327, 168.631, 56.554, -173.676]
  Call Extruder(907.934)
  MoveL 1492 to (52.45, 41.12, 8.6) mm, rotated rx 0 ry 90 rz 0 deg; joints [-9.348, 3.677, 52.398, 168.779, 56.585, -173.765]
  Call Extruder(908.789)
  MoveL 1493 to (58.88, 41.12, 8.6) mm, rotated rx 0 ry 90 rz 0 deg; joints [-9.282, 4.22, 50.906, 168.733, 55.647, -173.586]
  MoveL 1494 to (59.08, 41.12, 8.6) mm, rotated rx 0 ry 90 rz 0 deg; joints [-9.28, 4.238, 50.858, 168.732, 55.618, -173.58]
  Set speed (120.0 mm/s)
  MoveL 1495 to (57.59, 48.31, 8.6) mm, rotated rx 0 ry 90 rz 0 deg; joints [-9.744, 4.213, 50.925, 168.18, 55.712, -173.276]
  Set speed (1000.0 mm/s)
  MoveL 1496 to (57.66, 48.38, 8.6) mm, rotated rx 0 ry 90 rz 0 deg; joints [-9.747, 4.22, 50.906, 168.174, 55.701, -173.271]
  Set speed (30.0 mm/s)
  Call Extruder(908.842)
  MoveL 1497 to (57.66, 48.78, 8.6) mm, rotated rx 0 ry 90 rz 0 deg; joints [-9.772, 4.226, 50.89, 168.142, 55.694, -173.251]
  Call Extruder(909.119)
  MoveL 1498 to (57.66, 50.86, 8.6) mm, rotated rx 0 ry 90 rz 0 deg; joints [-9.902, 4.258, 50.804, 167.979, 55.656, -173.15]
  Call Extruder(909.377)
  MoveL 1499 to (59.6, 50.86, 8.6) mm, rotated rx 0 ry 90 rz 0 deg; joints [-9.881, 4.426, 50.345, 167.963, 55.37, -173.091]
  Call Extruder(910.539)
  MoveL 1500 to (59.6, 59.6, 8.6) mm, rotated rx 0 ry 90 rz 0 deg; joints [-10.423, 4.564, 49.972, 167.274, 55.206, -172.657]
  Call Extruder(913.094)
  MoveL 1501 to (40.4, 59.6, 8.6) mm, rotated rx 0 ry 90 rz 0 deg; joints [-10.646, 2.973, 54.364, 167.413, 57.967, -173.246]
  Call Extruder(915.648)
  MoveL 1502 to (40.4, 40.4, 8.6) mm, rotated rx 0 ry 90 rz 0 deg; joints [-9.429, 2.711, 55.104, 168.899, 58.301, -174.114]
  Call Extruder(916.561)
  MoveL 1503 to (47.26, 40.4, 8.6) mm, rotated rx 0 ry 90 rz 0 deg; joints [-9.357, 3.246, 53.597, 168.865, 57.339, -173.937]
  Call Extruder(916.813)
  MoveL 1504 to (47.26, 42.3, 8.6) mm, rotated rx 0 ry 90 rz 0 deg; joints [-9.476, 3.271, 53.526, 168.718, 57.308, -173.85]
  Call Extruder(917.407)
  MoveL 1505 to (51.73, 42.3, 8.6) mm, rotated rx 0 ry 90 rz 0 deg; joints [-9.43, 3.634, 52.518, 168.692, 56.669, -173.73]
  Call Extruder(917.659)
  MoveL 1506 to (51.73, 40.4, 8.6) mm, rotated rx 0 ry 90 rz 0 deg; joints [-9.31, 3.608, 52.589, 168.839, 56.701, -173.818]
  Call Extruder(918.706)
  MoveL 1507 to (59.6, 40.4, 8.6) mm, rotated rx 0 ry 90 rz 0 deg; joints [-9.23, 4.273, 50.763, 168.784, 55.553, -173.6]
  Call Extruder(919.768)
  MoveL 1508 to (59.6, 48.38, 8.6) mm, rotated rx 0 ry 90 rz 0 deg; joints [-9.727, 4.389, 50.448, 168.158, 55.414, -173.213]
  Call Extruder(919.972)
  MoveL 1509 to (58.06, 48.38, 8.6) mm, rotated rx 0 ry 90 rz 0 deg; joints [-9.743, 4.255, 50.812, 168.171, 55.642, -173.259]
  Call Extruder(920.007)
  MoveL 1510 to (57.66, 48.38, 8.6) mm, rotated rx 0 ry 90 rz 0 deg; joints [-9.747, 4.22, 50.906, 168.174, 55.701, -173.271]
  Set speed (120.0 mm/s)
  MoveL 1511 to (57.66, 48.78, 8.6) mm, rotated rx 0 ry 90 rz 0 deg; joints [-9.772, 4.226, 50.89, 168.142, 55.694, -173.251]
  Set speed (1000.0 mm/s)
  MoveL 1512 to (56.86, 48.78, 8.6) mm, rotated rx 0 ry 90 rz 0 deg; joints [-9.781, 4.157, 51.078, 168.149, 55.811, -173.275]
  MoveL 1513 to (52.43, 41.12, 8.6) mm, rotated rx 0 ry 90 rz 0 deg; joints [-9.348, 3.676, 52.402, 168.779, 56.588, -173.765]
  MoveL 1514 to (52.43, 41.12, 9) mm, rotated rx 0 ry 90 rz 0 deg; joints [-9.348, 3.633, 52.449, 168.779, 56.592, -173.766]
  Set speed (60.0 mm/s)
  Call Extruder(921.219)
  MoveL 1515 to (58.88, 47.57, 9) mm, rotated rx 0 ry 90 rz 0 deg; joints [-9.684, 4.27, 50.7, 168.228, 55.54, -173.275]
  Call Extruder(922.077)
  MoveL 1516 to (58.88, 41.12, 9) mm, rotated rx 0 ry 90 rz 0 deg; joints [-9.282, 4.177, 50.954, 168.734, 55.652, -173.587]
  Call Extruder(925.419)
  MoveL 1517 to (41.12, 58.88, 9) mm, rotated rx 0 ry 90 rz 0 deg; joints [-10.592, 2.976, 54.282, 167.466, 57.883, -173.259]
  Call Extruder(925.419)
  MoveL 1518 to (41.12, 58.88, 9) mm, rotated rx 0 ry 90 rz 0 deg; joints [-10.592, 2.976, 54.282, 167.466, 57.883, -173.259]
  Call Extruder(926.276)
  MoveL 1519 to (41.12, 52.43, 9) mm, rotated rx 0 ry 90 rz 0 deg; joints [-10.184, 2.884, 54.541, 167.966, 57.999, -173.554]
  Call Extruder(927.489)
  MoveL 1520 to (47.56, 58.88, 9) mm, rotated rx 0 ry 90 rz 0 deg; joints [-10.516, 3.488, 52.848, 167.427, 56.975, -173.069]
  Call Extruder(928.137)
  MoveL 1521 to (52.43, 58.88, 9) mm, rotated rx 0 ry 90 rz 0 deg; joints [-10.46, 3.891, 51.737, 167.392, 56.276, -172.921]
  Call Extruder(929.350)
  MoveL 1522 to (58.88, 52.43, 9) mm, rotated rx 0 ry 90 rz 0 deg; joints [-9.986, 4.343, 50.5, 167.846, 55.452, -173.037]
  Call Extruder(930.207)
  MoveL 1523 to (58.88, 58.88, 9) mm, rotated rx 0 ry 90 rz 0 deg; joints [-10.386, 4.445, 50.224, 167.338, 55.332, -172.717]
  Call Extruder(930.208)
  MoveL 1524 to (58.88, 58.88, 9) mm, rotated rx 0 ry 90 rz 0 deg; joints [-10.386, 4.445, 50.224, 167.338, 55.332, -172.717]
  Call Extruder(933.549)
  MoveL 1525 to (41.12, 41.12, 9) mm, rotated rx 0 ry 90 rz 0 deg; joints [-9.467, 2.733, 54.967, 168.84, 58.192, -174.064]
  Call Extruder(934.407)
  MoveL 1526 to (41.12, 47.56, 9) mm, rotated rx 0 ry 90 rz 0 deg; joints [-9.876, 2.817, 54.729, 168.342, 58.084, -173.775]
  Call Extruder(935.469)
  MoveL 1527 to (46.76, 41.92, 9) mm, rotated rx 0 ry 90 rz 0 deg; joints [-9.458, 3.184, 53.697, 168.75, 57.388, -173.881]
  Call Extruder(935.614)
  MoveL 1528 to (46.76, 43.02, 9) mm, rotated rx 0 ry 90 rz 0 deg; joints [-9.527, 3.199, 53.656, 168.665, 57.369, -173.831]
  Call Extruder(936.337)
  MoveL 1529 to (52.2, 43.02, 9) mm, rotated rx 0 ry 90 rz 0 deg; joints [-9.47, 3.639, 52.431, 168.633, 56.594, -173.684]
  Call Extruder(936.589)
  MoveL 1530 to (52.2, 41.12, 9) mm, rotated rx 0 ry 90 rz 0 deg; joints [-9.351, 3.613, 52.502, 168.781, 56.625, -173.773]
  Call Extruder(937.478)
  MoveL 1531 to (58.88, 41.12, 9) mm, rotated rx 0 ry 90 rz 0 deg; joints [-9.282, 4.177, 50.954, 168.734, 55.652, -173.587]
  MoveL 1532 to (59.08, 41.12, 9) mm, rotated rx 0 ry 90 rz 0 deg; joints [-9.28, 4.194, 50.907, 168.732, 55.622, -173.581]
  Set speed (120.0 mm/s)
  MoveL 1533 to (57.59, 48.3, 9) mm, rotated rx 0 ry 90 rz 0 deg; joints [-9.744, 4.17, 50.973, 168.181, 55.717, -173.277]
  Set speed (1000.0 mm/s)
  MoveL 1534 to (57.66, 48.37, 9) mm, rotated rx 0 ry 90 rz 0 deg; joints [-9.747, 4.177, 50.954, 168.175, 55.705, -173.272]
  Set speed (30.0 mm/s)
  Call Extruder(937.738)
  MoveL 1535 to (57.66, 50.32, 9) mm, rotated rx 0 ry 90 rz 0 deg; joints [-9.869, 4.206, 50.875, 168.022, 55.67, -173.177]
  Call Extruder(937.808)
  MoveL 1536 to (57.67, 50.85, 9) mm, rotated rx 0 ry 90 rz 0 deg; joints [-9.901, 4.214, 50.852, 167.98, 55.66, -173.151]
  Call Extruder(938.065)
  MoveL 1537 to (59.6, 50.86, 9) mm, rotated rx 0 ry 90 rz 0 deg; joints [-9.881, 4.382, 50.394, 167.964, 55.374, -173.092]
  Call Extruder(939.229)
  MoveL 1538 to (59.6, 59.6, 9) mm, rotated rx 0 ry 90 rz 0 deg; joints [-10.423, 4.52, 50.02, 167.274, 55.211, -172.658]
  Call Extruder(941.783)
  MoveL 1539 to (40.4, 59.6, 9) mm, rotated rx 0 ry 90 rz 0 deg; joints [-10.646, 2.93, 54.41, 167.414, 57.97, -173.247]
  Call Extruder(944.338)
  MoveL 1540 to (40.4, 40.4, 9) mm, rotated rx 0 ry 90 rz 0 deg; joints [-9.429, 2.669, 55.149, 168.899, 58.304, -174.114]
  Call Extruder(945.280)
  MoveL 1541 to (47.48, 40.4, 9) mm, rotated rx 0 ry 90 rz 0 deg; joints [-9.354, 3.221, 53.593, 168.864, 57.311, -173.932]
  Call Extruder(945.532)
  MoveL 1542 to (47.48, 42.3, 9) mm, rotated rx 0 ry 90 rz 0 deg; joints [-9.474, 3.246, 53.522, 168.717, 57.279, -173.845]
  Call Extruder(946.063)
  MoveL 1543 to (51.48, 42.3, 9) mm, rotated rx 0 ry 90 rz 0 deg; joints [-9.432, 3.57, 52.622, 168.694, 56.709, -173.737]
  Call Extruder(946.316)
  MoveL 1544 to (51.48, 40.4, 9) mm, rotated rx 0 ry 90 rz 0 deg; joints [-9.313, 3.544, 52.693, 168.841, 56.741, -173.826]
  Call Extruder(947.396)
  MoveL 1545 to (59.6, 40.4, 9) mm, rotated rx 0 ry 90 rz 0 deg; joints [-9.23, 4.229, 50.812, 168.785, 55.557, -173.601]
  Call Extruder(948.457)
  MoveL 1546 to (59.6, 48.37, 9) mm, rotated rx 0 ry 90 rz 0 deg; joints [-9.726, 4.345, 50.496, 168.159, 55.419, -173.214]
  Call Extruder(948.715)
  MoveL 1547 to (57.66, 48.37, 9) mm, rotated rx 0 ry 90 rz 0 deg; joints [-9.747, 4.177, 50.954, 168.175, 55.705, -173.272]
  Set speed (120.0 mm/s)
  MoveL 1548 to (57.66, 48.77, 9) mm, rotated rx 0 ry 90 rz 0 deg; joints [-9.772, 4.183, 50.938, 168.143, 55.698, -173.252]
  Set speed (1000.0 mm/s)
  MoveL 1549 to (56.86, 48.77, 9) mm, rotated rx 0 ry 90 rz 0 deg; joints [-9.781, 4.114, 51.126, 168.15, 55.816, -173.276]
  MoveL 1550 to (52.43, 41.12, 9) mm, rotated rx 0 ry 90 rz 0 deg; joints [-9.348, 3.633, 52.449, 168.779, 56.592, -173.766]
  MoveL 1551 to (52.43, 41.12, 9.4) mm, rotated rx 0 ry 90 rz 0 deg; joints [-9.348, 3.589, 52.496, 168.78, 56.595, -173.767]
  Set speed (60.0 mm/s)
  Call Extruder(949.928)
  MoveL 1552 to (58.88, 47.56, 9.4) mm, rotated rx 0 ry 90 rz 0 deg; joints [-9.684, 4.226, 50.748, 168.229, 55.544, -173.276]
  Call Extruder(950.785)
  MoveL 1553 to (58.88, 41.12, 9.4) mm, rotated rx 0 ry 90 rz 0 deg; joints [-9.282, 4.133, 51.002, 168.735, 55.656, -173.588]
  Call Extruder(954.127)
  MoveL 1554 to (41.12, 58.88, 9.4) mm, rotated rx 0 ry 90 rz 0 deg; joints [-10.592, 2.933, 54.328, 167.466, 57.886, -173.26]
  Call Extruder(954.127)
  MoveL 1555 to (41.12, 58.88, 9.4) mm, rotated rx 0 ry 90 rz 0 deg; joints [-10.592, 2.933, 54.327, 167.466, 57.886, -173.26]
  Call Extruder(954.984)
  MoveL 1556 to (41.12, 52.43, 9.4) mm, rotated rx 0 ry 90 rz 0 deg; joints [-10.184, 2.841, 54.586, 167.966, 58.002, -173.555]
  Call Extruder(956.197)
  MoveL 1557 to (47.57, 58.88, 9.4) mm, rotated rx 0 ry 90 rz 0 deg; joints [-10.516, 3.445, 52.895, 167.427, 56.979, -173.07]
  Call Extruder(956.845)
  MoveL 1558 to (52.43, 58.88, 9.4) mm, rotated rx 0 ry 90 rz 0 deg; joints [-10.46, 3.847, 51.784, 167.393, 56.28, -172.922]
  Call Extruder(958.056)
  MoveL 1559 to (58.87, 52.44, 9.4) mm, rotated rx 0 ry 90 rz 0 deg; joints [-9.987, 4.299, 50.55, 167.846, 55.458, -173.038]
  Call Extruder(958.913)
  MoveL 1560 to (58.88, 58.88, 9.4) mm, rotated rx 0 ry 90 rz 0 deg; joints [-10.386, 4.401, 50.273, 167.339, 55.337, -172.719]
  Call Extruder(958.913)
  MoveL 1561 to (58.88, 58.88, 9.4) mm, rotated rx 0 ry 90 rz 0 deg; joints [-10.386, 4.401, 50.273, 167.339, 55.337, -172.719]
  Call Extruder(962.254)
  MoveL 1562 to (41.12, 41.12, 9.4) mm, rotated rx 0 ry 90 rz 0 deg; joints [-9.467, 2.691, 55.013, 168.841, 58.195, -174.065]
  Call Extruder(963.112)
  MoveL 1563 to (41.12, 47.57, 9.4) mm, rotated rx 0 ry 90 rz 0 deg; joints [-9.876, 2.775, 54.774, 168.343, 58.087, -173.776]
  Call Extruder(964.216)
  MoveL 1564 to (46.99, 41.7, 9.4) mm, rotated rx 0 ry 90 rz 0 deg; joints [-9.442, 3.156, 53.702, 168.767, 57.363, -173.886]
  Call Extruder(964.391)
  MoveL 1565 to (46.99, 43.02, 9.4) mm, rotated rx 0 ry 90 rz 0 deg; joints [-9.525, 3.174, 53.652, 168.665, 57.341, -173.826]
  Call Extruder(965.050)
  MoveL 1566 to (51.94, 43.02, 9.4) mm, rotated rx 0 ry 90 rz 0 deg; joints [-9.473, 3.575, 52.535, 168.635, 56.634, -173.692]
  Call Extruder(965.303)
  MoveL 1567 to (51.95, 41.12, 9.4) mm, rotated rx 0 ry 90 rz 0 deg; joints [-9.354, 3.549, 52.607, 168.783, 56.665, -173.78]
  Call Extruder(966.225)
  MoveL 1568 to (58.88, 41.12, 9.4) mm, rotated rx 0 ry 90 rz 0 deg; joints [-9.282, 4.133, 51.002, 168.734, 55.656, -173.588]
  MoveL 1569 to (59.08, 41.12, 9.4) mm, rotated rx 0 ry 90 rz 0 deg; joints [-9.28, 4.15, 50.955, 168.733, 55.626, -173.582]
  Set speed (120.0 mm/s)
  MoveL 1570 to (51.29, 42.37, 9.4) mm, rotated rx 0 ry 90 rz 0 deg; joints [-9.439, 3.513, 52.708, 168.69, 56.738, -173.74]
  Set speed (1000.0 mm/s)
  MoveL 1571 to (51.22, 42.3, 9.4) mm, rotated rx 0 ry 90 rz 0 deg; joints [-9.435, 3.506, 52.726, 168.696, 56.749, -173.745]
  Set speed (30.0 mm/s)
  Call Extruder(966.477)
  MoveL 1572 to (51.23, 40.4, 9.4) mm, rotated rx 0 ry 90 rz 0 deg; joints [-9.316, 3.481, 52.797, 168.843, 56.78, -173.833]
  Call Extruder(967.591)
  MoveL 1573 to (59.6, 40.4, 9.4) mm, rotated rx 0 ry 90 rz 0 deg; joints [-9.23, 4.185, 50.86, 168.785, 55.562, -173.602]
  Call Extruder(968.651)
  MoveL 1574 to (59.6, 48.36, 9.4) mm, rotated rx 0 ry 90 rz 0 deg; joints [-9.726, 4.301, 50.545, 168.161, 55.424, -173.216]
  Call Extruder(968.908)
  MoveL 1575 to (57.66, 48.37, 9.4) mm, rotated rx 0 ry 90 rz 0 deg; joints [-9.747, 4.133, 51.002, 168.176, 55.709, -173.273]
  Call Extruder(969.236)
  MoveL 1576 to (57.66, 50.84, 9.4) mm, rotated rx 0 ry 90 rz 0 deg; joints [-9.901, 4.17, 50.902, 167.982, 55.665, -173.153]
  Call Extruder(969.493)
  MoveL 1577 to (59.59, 50.85, 9.4) mm, rotated rx 0 ry 90 rz 0 deg; joints [-9.88, 4.338, 50.445, 167.965, 55.38, -173.094]
  Call Extruder(970.604)
  MoveL 1578 to (59.6, 59.2, 9.4) mm, rotated rx 0 ry 90 rz 0 deg; joints [-10.398, 4.47, 50.087, 167.307, 55.224, -172.679]
  Call Extruder(970.657)
  MoveL 1579 to (59.6, 59.6, 9.4) mm, rotated rx 0 ry 90 rz 0 deg; joints [-10.423, 4.476, 50.069, 167.275, 55.216, -172.659]
  Call Extruder(970.692)
  MoveL 1580 to (59.2, 59.6, 9.4) mm, rotated rx 0 ry 90 rz 0 deg; joints [-10.427, 4.441, 50.165, 167.279, 55.275, -172.672]
  Call Extruder(973.193)
  MoveL 1581 to (40.4, 59.6, 9.4) mm, rotated rx 0 ry 90 rz 0 deg; joints [-10.646, 2.888, 54.455, 167.414, 57.973, -173.247]
  Call Extruder(975.747)
  MoveL 1582 to (40.4, 40.4, 9.4) mm, rotated rx 0 ry 90 rz 0 deg; joints [-9.429, 2.627, 55.194, 168.899, 58.307, -174.115]
  Call Extruder(976.719)
  MoveL 1583 to (47.71, 40.4, 9.4) mm, rotated rx 0 ry 90 rz 0 deg; joints [-9.352, 3.196, 53.589, 168.864, 57.283, -173.927]
  Call Extruder(976.971)
  MoveL 1584 to (47.71, 42.3, 9.4) mm, rotated rx 0 ry 90 rz 0 deg; joints [-9.472, 3.221, 53.519, 168.716, 57.251, -173.84]
  Call Extruder(977.439)
  MoveL 1585 to (51.22, 42.3, 9.4) mm, rotated rx 0 ry 90 rz 0 deg; joints [-9.435, 3.506, 52.726, 168.696, 56.749, -173.745]
  Set speed (120.0 mm/s)
  MoveL 1586 to (51.23, 41.9, 9.4) mm, rotated rx 0 ry 90 rz 0 deg; joints [-9.41, 3.501, 52.741, 168.727, 56.756, -173.764]
  Set speed (1000.0 mm/s)
  MoveL 1587 to (52.02, 41.9, 9.4) mm, rotated rx 0 ry 90 rz 0 deg; joints [-9.401, 3.566, 52.559, 168.722, 56.641, -173.742]
  MoveL 1588 to (52.43, 41.12, 9.4) mm, rotated rx 0 ry 90 rz 0 deg; joints [-9.348, 3.589, 52.496, 168.78, 56.595, -173.767]
  MoveL 1589 to (52.43, 41.12, 9.8) mm, rotated rx 0 ry 90 rz 0 deg; joints [-9.348, 3.546, 52.542, 168.78, 56.599, -173.768]
  Set speed (60.0 mm/s)
  Call Extruder(978.624)
  MoveL 1590 to (58.73, 47.42, 9.8) mm, rotated rx 0 ry 90 rz 0 deg; joints [-9.676, 4.168, 50.837, 168.242, 55.573, -173.289]
  Call Extruder(978.644)
  MoveL 1591 to (58.88, 47.42, 9.8) mm, rotated rx 0 ry 90 rz 0 deg; joints [-9.675, 4.181, 50.802, 168.241, 55.551, -173.284]
  Call Extruder(979.482)
  MoveL 1592 to (58.88, 41.12, 9.8) mm, rotated rx 0 ry 90 rz 0 deg; joints [-9.282, 4.09, 51.05, 168.735, 55.66, -173.589]
  Call Extruder(982.824)
  MoveL 1593 to (41.12, 58.88, 9.8) mm, rotated rx 0 ry 90 rz 0 deg; joints [-10.592, 2.89, 54.373, 167.467, 57.889, -173.261]
  Call Extruder(982.824)
  MoveL 1594 to (41.12, 58.88, 9.8) mm, rotated rx 0 ry 90 rz 0 deg; joints [-10.592, 2.891, 54.373, 167.466, 57.889, -173.261]
  Call Extruder(983.682)
  MoveL 1595 to (41.12, 52.43, 9.8) mm, rotated rx 0 ry 90 rz 0 deg; joints [-10.184, 2.799, 54.631, 167.966, 58.005, -173.556]
  Call Extruder(984.895)
  MoveL 1596 to (47.57, 58.88, 9.8) mm, rotated rx 0 ry 90 rz 0 deg; joints [-10.516, 3.403, 52.941, 167.428, 56.982, -173.071]
  Call Extruder(985.542)
  MoveL 1597 to (52.43, 58.88, 9.8) mm, rotated rx 0 ry 90 rz 0 deg; joints [-10.46, 3.804, 51.831, 167.393, 56.284, -172.923]
  Call Extruder(986.755)
  MoveL 1598 to (58.88, 52.43, 9.8) mm, rotated rx 0 ry 90 rz 0 deg; joints [-9.986, 4.256, 50.596, 167.847, 55.461, -173.039]
  Call Extruder(987.613)
  MoveL 1599 to (58.88, 58.88, 9.8) mm, rotated rx 0 ry 90 rz 0 deg; joints [-10.386, 4.357, 50.321, 167.339, 55.341, -172.72]
  Call Extruder(987.613)
  MoveL 1600 to (58.88, 58.88, 9.8) mm, rotated rx 0 ry 90 rz 0 deg; joints [-10.386, 4.357, 50.321, 167.339, 55.341, -172.72]
  Call Extruder(990.954)
  MoveL 1601 to (41.12, 41.12, 9.8) mm, rotated rx 0 ry 90 rz 0 deg; joints [-9.467, 2.648, 55.058, 168.841, 58.198, -174.065]
  Call Extruder(991.812)
  MoveL 1602 to (41.12, 47.57, 9.8) mm, rotated rx 0 ry 90 rz 0 deg; joints [-9.876, 2.732, 54.819, 168.343, 58.09, -173.776]
  Call Extruder(992.958)
  MoveL 1603 to (47.21, 41.48, 9.8) mm, rotated rx 0 ry 90 rz 0 deg; joints [-9.425, 3.128, 53.706, 168.783, 57.338, -173.891]
  Call Extruder(993.163)
  MoveL 1604 to (47.21, 43.02, 9.8) mm, rotated rx 0 ry 90 rz 0 deg; joints [-9.522, 3.149, 53.648, 168.664, 57.312, -173.821]
  Call Extruder(993.758)
  MoveL 1605 to (51.69, 43.02, 9.8) mm, rotated rx 0 ry 90 rz 0 deg; joints [-9.475, 3.511, 52.64, 168.637, 56.674, -173.699]
  Call Extruder(994.011)
  MoveL 1606 to (51.69, 41.12, 9.8) mm, rotated rx 0 ry 90 rz 0 deg; joints [-9.356, 3.485, 52.711, 168.785, 56.705, -173.788]
  Call Extruder(994.967)
  MoveL 1607 to (58.88, 41.12, 9.8) mm, rotated rx 0 ry 90 rz 0 deg; joints [-9.282, 4.09, 51.05, 168.735, 55.66, -173.589]
  MoveL 1608 to (59.08, 41.12, 9.8) mm, rotated rx 0 ry 90 rz 0 deg; joints [-9.28, 4.107, 51.002, 168.734, 55.631, -173.583]
  Set speed (120.0 mm/s)
  MoveL 1609 to (57.64, 48.11, 9.8) mm, rotated rx 0 ry 90 rz 0 deg; joints [-9.731, 4.083, 51.067, 168.197, 55.722, -173.287]
  Set speed (1000.0 mm/s)
  MoveL 1610 to (57.59, 51.13, 9.8) mm, rotated rx 0 ry 90 rz 0 deg; joints [-9.919, 4.124, 50.955, 167.961, 55.675, -173.142]
  MoveL 1611 to (57.66, 51.06, 9.8) mm, rotated rx 0 ry 90 rz 0 deg; joints [-9.914, 4.129, 50.941, 167.965, 55.666, -173.144]
  Set speed (30.0 mm/s)
  Call Extruder(995.225)
  MoveL 1612 to (59.6, 51.06, 9.8) mm, rotated rx 0 ry 90 rz 0 deg; joints [-9.893, 4.298, 50.482, 167.949, 55.38, -173.084]
  Call Extruder(996.361)
  MoveL 1613 to (59.6, 59.6, 9.8) mm, rotated rx 0 ry 90 rz 0 deg; joints [-10.423, 4.433, 50.118, 167.276, 55.221, -172.661]
  Call Extruder(998.916)
  MoveL 1614 to (40.4, 59.6, 9.8) mm, rotated rx 0 ry 90 rz 0 deg; joints [-10.646, 2.845, 54.501, 167.414, 57.976, -173.248]
  Call Extruder(1001.470)
  MoveL 1615 to (40.4, 40.4, 9.8) mm, rotated rx 0 ry 90 rz 0 deg; joints [-9.429, 2.584, 55.239, 168.9, 58.309, -174.115]
  Call Extruder(1002.471)
  MoveL 1616 to (47.93, 40.4, 9.8) mm, rotated rx 0 ry 90 rz 0 deg; joints [-9.35, 3.171, 53.586, 168.863, 57.254, -173.922]
  Call Extruder(1002.724)
  MoveL 1617 to (47.93, 42.3, 9.8) mm, rotated rx 0 ry 90 rz 0 deg; joints [-9.469, 3.196, 53.515, 168.716, 57.222, -173.835]
  Call Extruder(1003.128)
  MoveL 1618 to (50.97, 42.3, 9.8) mm, rotated rx 0 ry 90 rz 0 deg; joints [-9.438, 3.442, 52.83, 168.698, 56.789, -173.753]
  Call Extruder(1003.381)
  MoveL 1619 to (50.97, 40.4, 9.8) mm, rotated rx 0 ry 90 rz 0 deg; joints [-9.318, 3.417, 52.901, 168.845, 56.82, -173.841]
  Call Extruder(1004.528)
  MoveL 1620 to (59.6, 40.4, 9.8) mm, rotated rx 0 ry 90 rz 0 deg; joints [-9.23, 4.142, 50.908, 168.786, 55.566, -173.603]
  Call Extruder(1005.558)
  MoveL 1621 to (59.6, 48.14, 9.8) mm, rotated rx 0 ry 90 rz 0 deg; joints [-9.712, 4.254, 50.602, 168.179, 55.432, -173.228]
  Call Extruder(1005.815)
  MoveL 1622 to (57.66, 48.14, 9.8) mm, rotated rx 0 ry 90 rz 0 deg; joints [-9.733, 4.086, 51.059, 168.194, 55.717, -173.285]
  Call Extruder(1006.203)
  MoveL 1623 to (57.66, 51.06, 9.8) mm, rotated rx 0 ry 90 rz 0 deg; joints [-9.914, 4.129, 50.941, 167.965, 55.666, -173.144]
  Set speed (120.0 mm/s)
  MoveL 1624 to (58.06, 51.06, 9.8) mm, rotated rx 0 ry 90 rz 0 deg; joints [-9.91, 4.164, 50.847, 167.962, 55.607, -173.132]
  Set speed (1000.0 mm/s)
  MoveL 1625 to (58.06, 51.86, 9.8) mm, rotated rx 0 ry 90 rz 0 deg; joints [-9.96, 4.176, 50.814, 167.899, 55.593, -173.092]
  MoveL 1626 to (52.43, 41.12, 9.8) mm, rotated rx 0 ry 90 rz 0 deg; joints [-9.348, 3.546, 52.542, 168.78, 56.599, -173.768]
  MoveL 1627 to (52.43, 41.12, 10.2) mm, rotated rx 0 ry 90 rz 0 deg; joints [-9.348, 3.503, 52.589, 168.781, 56.602, -173.769]
  Set speed (60.0 mm/s)
  Call Extruder(1007.343)
  MoveL 1628 to (58.49, 47.18, 10.2) mm, rotated rx 0 ry 90 rz 0 deg; joints [-9.664, 4.1, 50.951, 168.264, 55.617, -173.309]
  Call Extruder(1007.395)
  MoveL 1629 to (58.88, 47.18, 10.2) mm, rotated rx 0 ry 90 rz 0 deg; joints [-9.66, 4.133, 50.859, 168.261, 55.56, -173.297]
  Call Extruder(1008.201)
  MoveL 1630 to (58.88, 41.12, 10.2) mm, rotated rx 0 ry 90 rz 0 deg; joints [-9.282, 4.046, 51.098, 168.736, 55.665, -173.59]
  Call Extruder(1011.543)
  MoveL 1631 to (41.12, 58.88, 10.2) mm, rotated rx 0 ry 90 rz 0 deg; joints [-10.592, 2.848, 54.419, 167.467, 57.892, -173.261]
  Call Extruder(1011.543)
  MoveL 1632 to (41.12, 58.88, 10.2) mm, rotated rx 0 ry 90 rz 0 deg; joints [-10.592, 2.848, 54.418, 167.467, 57.892, -173.261]
  Call Extruder(1012.401)
  MoveL 1633 to (41.12, 52.43, 10.2) mm, rotated rx 0 ry 90 rz 0 deg; joints [-10.184, 2.756, 54.677, 167.967, 58.008, -173.557]
  Call Extruder(1013.613)
  MoveL 1634 to (47.57, 58.88, 10.2) mm, rotated rx 0 ry 90 rz 0 deg; joints [-10.516, 3.36, 52.987, 167.428, 56.985, -173.072]
  Call Extruder(1014.261)
  MoveL 1635 to (52.43, 58.88, 10.2) mm, rotated rx 0 ry 90 rz 0 deg; joints [-10.46, 3.761, 51.879, 167.394, 56.288, -172.924]
  Call Extruder(1015.474)
  MoveL 1636 to (58.88, 52.43, 10.2) mm, rotated rx 0 ry 90 rz 0 deg; joints [-9.986, 4.212, 50.645, 167.848, 55.466, -173.04]
  Call Extruder(1016.331)
  MoveL 1637 to (58.88, 58.88, 10.2) mm, rotated rx 0 ry 90 rz 0 deg; joints [-10.386, 4.314, 50.369, 167.34, 55.346, -172.721]
  Call Extruder(1016.331)
  MoveL 1638 to (58.88, 58.88, 10.2) mm, rotated rx 0 ry 90 rz 0 deg; joints [-10.386, 4.314, 50.37, 167.34, 55.346, -172.721]
  Call Extruder(1019.673)
  MoveL 1639 to (41.12, 41.12, 10.2) mm, rotated rx 0 ry 90 rz 0 deg; joints [-9.467, 2.606, 55.103, 168.841, 58.2, -174.066]
  Call Extruder(1020.530)
  MoveL 1640 to (41.12, 47.56, 10.2) mm, rotated rx 0 ry 90 rz 0 deg; joints [-9.876, 2.69, 54.864, 168.343, 58.092, -173.777]
  Call Extruder(1021.718)
  MoveL 1641 to (47.43, 41.26, 10.2) mm, rotated rx 0 ry 90 rz 0 deg; joints [-9.409, 3.1, 53.712, 168.8, 57.314, -173.896]
  Call Extruder(1021.947)
  MoveL 1642 to (47.43, 42.98, 10.2) mm, rotated rx 0 ry 90 rz 0 deg; joints [-9.518, 3.123, 53.647, 168.666, 57.285, -173.817]
  Call Extruder(1022.476)
  MoveL 1643 to (51.4, 43.03, 10.2) mm, rotated rx 0 ry 90 rz 0 deg; joints [-9.479, 3.445, 52.751, 168.638, 56.718, -173.708]
  Call Extruder(1022.730)
  MoveL 1644 to (51.43, 41.12, 10.2) mm, rotated rx 0 ry 90 rz 0 deg; joints [-9.359, 3.421, 52.818, 168.787, 56.747, -173.796]
  Call Extruder(1023.722)
  MoveL 1645 to (58.88, 41.12, 10.2) mm, rotated rx 0 ry 90 rz 0 deg; joints [-9.282, 4.046, 51.097, 168.736, 55.664, -173.59]
  MoveL 1646 to (59.08, 41.12, 10.2) mm, rotated rx 0 ry 90 rz 0 deg; joints [-9.28, 4.063, 51.05, 168.734, 55.635, -173.585]
  Set speed (120.0 mm/s)
  MoveL 1647 to (50.76, 42.37, 10.2) mm, rotated rx 0 ry 90 rz 0 deg; joints [-9.445, 3.383, 52.922, 168.693, 56.821, -173.756]
  Set speed (1000.0 mm/s)
  MoveL 1648 to (50.69, 42.3, 10.2) mm, rotated rx 0 ry 90 rz 0 deg; joints [-9.441, 3.377, 52.94, 168.699, 56.832, -173.761]
  Set speed (30.0 mm/s)
  Call Extruder(1023.975)
  MoveL 1649 to (50.72, 40.4, 10.2) mm, rotated rx 0 ry 90 rz 0 deg; joints [-9.321, 3.353, 53.006, 168.847, 56.861, -173.849]
  Call Extruder(1025.157)
  MoveL 1650 to (59.6, 40.4, 10.2) mm, rotated rx 0 ry 90 rz 0 deg; joints [-9.23, 4.098, 50.955, 168.786, 55.57, -173.604]
  Call Extruder(1026.154)
  MoveL 1651 to (59.6, 47.9, 10.2) mm, rotated rx 0 ry 90 rz 0 deg; joints [-9.697, 4.207, 50.66, 168.198, 55.441, -173.241]
  Call Extruder(1026.412)
  MoveL 1652 to (57.66, 47.9, 10.2) mm, rotated rx 0 ry 90 rz 0 deg; joints [-9.718, 4.039, 51.116, 168.214, 55.726, -173.298]
  Call Extruder(1026.862)
  MoveL 1653 to (57.66, 51.28, 10.2) mm, rotated rx 0 ry 90 rz 0 deg; joints [-9.928, 4.09, 50.979, 167.948, 55.666, -173.134]
  Call Extruder(1027.120)
  MoveL 1654 to (59.6, 51.29, 10.2) mm, rotated rx 0 ry 90 rz 0 deg; joints [-9.907, 4.258, 50.521, 167.932, 55.38, -173.074]
  Call Extruder(1028.226)
  MoveL 1655 to (59.6, 59.6, 10.2) mm, rotated rx 0 ry 90 rz 0 deg; joints [-10.423, 4.389, 50.166, 167.277, 55.225, -172.662]
  Call Extruder(1030.780)
  MoveL 1656 to (40.4, 59.6, 10.2) mm, rotated rx 0 ry 90 rz 0 deg; joints [-10.646, 2.803, 54.546, 167.415, 57.978, -173.249]
  Call Extruder(1033.334)
  MoveL 1657 to (40.4, 40.4, 10.2) mm, rotated rx 0 ry 90 rz 0 deg; joints [-9.429, 2.542, 55.284, 168.9, 58.312, -174.116]
  Call Extruder(1034.365)
  MoveL 1658 to (48.15, 40.4, 10.2) mm, rotated rx 0 ry 90 rz 0 deg; joints [-9.348, 3.146, 53.582, 168.862, 57.226, -173.917]
  Call Extruder(1034.614)
  MoveL 1659 to (48.15, 42.27, 10.2) mm, rotated rx 0 ry 90 rz 0 deg; joints [-9.466, 3.171, 53.513, 168.717, 57.195, -173.831]
  Call Extruder(1034.953)
  MoveL 1660 to (50.69, 42.3, 10.2) mm, rotated rx 0 ry 90 rz 0 deg; joints [-9.441, 3.377, 52.94, 168.699, 56.832, -173.761]
  Set speed (120.0 mm/s)
  MoveL 1661 to (50.7, 41.9, 10.2) mm, rotated rx 0 ry 90 rz 0 deg; joints [-9.416, 3.372, 52.954, 168.731, 56.838, -173.779]
  Set speed (1000.0 mm/s)
  MoveL 1662 to (51.5, 41.91, 10.2) mm, rotated rx 0 ry 90 rz 0 deg; joints [-9.408, 3.437, 52.772, 168.725, 56.724, -173.757]
  MoveL 1663 to (52.43, 41.12, 10.2) mm, rotated rx 0 ry 90 rz 0 deg; joints [-9.348, 3.503, 52.589, 168.781, 56.602, -173.769]
  MoveL 1664 to (52.43, 41.12, 10.6) mm, rotated rx 0 ry 90 rz 0 deg; joints [-9.348, 3.46, 52.635, 168.781, 56.606, -173.77]
  Set speed (60.0 mm/s)
  Call Extruder(1036.048)
  MoveL 1665 to (58.25, 46.94, 10.6) mm, rotated rx 0 ry 90 rz 0 deg; joints [-9.652, 4.032, 51.064, 168.285, 55.66, -173.328]
  Call Extruder(1036.131)
  MoveL 1666 to (58.88, 46.94, 10.6) mm, rotated rx 0 ry 90 rz 0 deg; joints [-9.645, 4.086, 50.917, 168.28, 55.568, -173.31]
  Call Extruder(1036.905)
  MoveL 1667 to (58.88, 41.12, 10.6) mm, rotated rx 0 ry 90 rz 0 deg; joints [-9.282, 4.003, 51.145, 168.736, 55.669, -173.591]
  Call Extruder(1040.247)
  MoveL 1668 to (41.12, 58.88, 10.6) mm, rotated rx 0 ry 90 rz 0 deg; joints [-10.592, 2.805, 54.464, 167.467, 57.894, -173.262]
  Call Extruder(1040.247)
  MoveL 1669 to (41.12, 58.88, 10.6) mm, rotated rx 0 ry 90 rz 0 deg; joints [-10.592, 2.805, 54.464, 167.467, 57.894, -173.262]
  Call Extruder(1041.105)
  MoveL 1670 to (41.12, 52.43, 10.6) mm, rotated rx 0 ry 90 rz 0 deg; joints [-10.184, 2.714, 54.722, 167.967, 58.01, -173.557]
  Call Extruder(1042.318)
  MoveL 1671 to (47.56, 58.88, 10.6) mm, rotated rx 0 ry 90 rz 0 deg; joints [-10.516, 3.317, 53.034, 167.429, 56.989, -173.073]
  Call Extruder(1042.965)
  MoveL 1672 to (52.43, 58.88, 10.6) mm, rotated rx 0 ry 90 rz 0 deg; joints [-10.46, 3.718, 51.926, 167.394, 56.292, -172.925]
  Call Extruder(1044.178)
  MoveL 1673 to (58.88, 52.43, 10.6) mm, rotated rx 0 ry 90 rz 0 deg; joints [-9.986, 4.169, 50.693, 167.848, 55.47, -173.041]
  Call Extruder(1045.036)
  MoveL 1674 to (58.88, 58.88, 10.6) mm, rotated rx 0 ry 90 rz 0 deg; joints [-10.386, 4.27, 50.418, 167.341, 55.35, -172.722]
  Call Extruder(1045.036)
  MoveL 1675 to (58.88, 58.88, 10.6) mm, rotated rx 0 ry 90 rz 0 deg; joints [-10.386, 4.27, 50.418, 167.341, 55.35, -172.722]
  Call Extruder(1048.377)
  MoveL 1676 to (41.12, 41.12, 10.6) mm, rotated rx 0 ry 90 rz 0 deg; joints [-9.467, 2.563, 55.148, 168.842, 58.203, -174.066]
  Call Extruder(1049.235)
  MoveL 1677 to (41.12, 47.56, 10.6) mm, rotated rx 0 ry 90 rz 0 deg; joints [-9.876, 2.648, 54.909, 168.344, 58.095, -173.778]
  Call Extruder(1050.393)
  MoveL 1678 to (47.28, 41.41, 10.6) mm, rotated rx 0 ry 90 rz 0 deg; joints [-9.42, 3.047, 53.786, 168.789, 57.336, -173.894]
  Call Extruder(1050.608)
  MoveL 1679 to (47.28, 43.02, 10.6) mm, rotated rx 0 ry 90 rz 0 deg; joints [-9.522, 3.068, 53.726, 168.664, 57.309, -173.82]
  Call Extruder(1051.192)
  MoveL 1680 to (51.67, 43.02, 10.6) mm, rotated rx 0 ry 90 rz 0 deg; joints [-9.476, 3.423, 52.738, 168.638, 56.684, -173.702]
  Call Extruder(1051.444)
  MoveL 1681 to (51.67, 41.12, 10.6) mm, rotated rx 0 ry 90 rz 0 deg; joints [-9.356, 3.398, 52.809, 168.786, 56.715, -173.79]
  Call Extruder(1052.404)
  MoveL 1682 to (58.88, 41.12, 10.6) mm, rotated rx 0 ry 90 rz 0 deg; joints [-9.282, 4.003, 51.145, 168.736, 55.669, -173.591]
  MoveL 1683 to (59.08, 41.12, 10.6) mm, rotated rx 0 ry 90 rz 0 deg; joints [-9.28, 4.02, 51.098, 168.735, 55.639, -173.586]
  Set speed (120.0 mm/s)
  MoveL 1684 to (50.98, 42.33, 10.6) mm, rotated rx 0 ry 90 rz 0 deg; joints [-9.439, 3.357, 52.921, 168.696, 56.794, -173.753]
  Set speed (1000.0 mm/s)
  MoveL 1685 to (47.93, 42.37, 10.6) mm, rotated rx 0 ry 90 rz 0 deg; joints [-9.474, 3.112, 53.605, 168.711, 57.228, -173.833]
  MoveL 1686 to (48, 42.3, 10.6) mm, rotated rx 0 ry 90 rz 0 deg; joints [-9.469, 3.116, 53.592, 168.716, 57.219, -173.834]
  Set speed (30.0 mm/s)
  Call Extruder(1052.457)
  MoveL 1687 to (48.4, 42.3, 10.6) mm, rotated rx 0 ry 90 rz 0 deg; joints [-9.465, 3.148, 53.503, 168.714, 57.163, -173.824]
  Call Extruder(1052.797)
  MoveL 1688 to (50.95, 42.3, 10.6) mm, rotated rx 0 ry 90 rz 0 deg; joints [-9.438, 3.355, 52.928, 168.699, 56.799, -173.755]
  Call Extruder(1053.049)
  MoveL 1689 to (50.95, 40.4, 10.6) mm, rotated rx 0 ry 90 rz 0 deg; joints [-9.319, 3.329, 52.999, 168.846, 56.83, -173.843]
  Call Extruder(1054.200)
  MoveL 1690 to (59.6, 40.4, 10.6) mm, rotated rx 0 ry 90 rz 0 deg; joints [-9.23, 4.055, 51.003, 168.787, 55.575, -173.605]
  Call Extruder(1055.165)
  MoveL 1691 to (59.6, 47.66, 10.6) mm, rotated rx 0 ry 90 rz 0 deg; joints [-9.682, 4.159, 50.718, 168.218, 55.449, -173.253]
  Call Extruder(1055.423)
  MoveL 1692 to (57.66, 47.66, 10.6) mm, rotated rx 0 ry 90 rz 0 deg; joints [-9.703, 3.992, 51.174, 168.233, 55.734, -173.311]
  Call Extruder(1055.935)
  MoveL 1693 to (57.66, 51.51, 10.6) mm, rotated rx 0 ry 90 rz 0 deg; joints [-9.942, 4.049, 51.017, 167.931, 55.666, -173.124]
  Call Extruder(1056.193)
  MoveL 1694 to (59.6, 51.51, 10.6) mm, rotated rx 0 ry 90 rz 0 deg; joints [-9.921, 4.218, 50.56, 167.915, 55.38, -173.064]
  Call Extruder(1057.268)
  MoveL 1695 to (59.6, 59.6, 10.6) mm, rotated rx 0 ry 90 rz 0 deg; joints [-10.423, 4.345, 50.215, 167.277, 55.23, -172.663]
  Call Extruder(1059.823)
  MoveL 1696 to (40.4, 59.6, 10.6) mm, rotated rx 0 ry 90 rz 0 deg; joints [-10.646, 2.76, 54.591, 167.415, 57.981, -173.25]
  Call Extruder(1062.377)
  MoveL 1697 to (40.4, 40.4, 10.6) mm, rotated rx 0 ry 90 rz 0 deg; joints [-9.429, 2.5, 55.329, 168.9, 58.314, -174.116]
  Call Extruder(1063.335)
  MoveL 1698 to (47.6, 40.4, 10.6) mm, rotated rx 0 ry 90 rz 0 deg; joints [-9.353, 3.059, 53.751, 168.865, 57.307, -173.932]
  Call Extruder(1063.388)
  MoveL 1699 to (48, 40.4, 10.6) mm, rotated rx 0 ry 90 rz 0 deg; joints [-9.349, 3.091, 53.662, 168.863, 57.251, -173.921]
  Call Extruder(1063.422)
  MoveL 1700 to (48, 40.8, 10.6) mm, rotated rx 0 ry 90 rz 0 deg; joints [-9.374, 3.096, 53.647, 168.832, 57.244, -173.903]
  Call Extruder(1063.568)
  MoveL 1701 to (48, 41.9, 10.6) mm, rotated rx 0 ry 90 rz 0 deg; joints [-9.444, 3.111, 53.607, 168.747, 57.226, -173.853]
  Call Extruder(1063.603)
  MoveL 1702 to (48, 42.3, 10.6) mm, rotated rx 0 ry 90 rz 0 deg; joints [-9.469, 3.116, 53.592, 168.716, 57.219, -173.834]
  Set speed (120.0 mm/s)
  MoveL 1703 to (48.4, 42.3, 10.6) mm, rotated rx 0 ry 90 rz 0 deg; joints [-9.465, 3.148, 53.503, 168.714, 57.163, -173.824]
  Set speed (1000.0 mm/s)
  MoveL 1704 to (48.4, 43.1, 10.6) mm, rotated rx 0 ry 90 rz 0 deg; joints [-9.515, 3.159, 53.473, 168.652, 57.149, -173.787]
  MoveL 1705 to (50.98, 42.33, 10.6) mm, rotated rx 0 ry 90 rz 0 deg; joints [-9.439, 3.357, 52.921, 168.696, 56.794, -173.753]
  MoveL 1706 to (52.43, 41.12, 10.6) mm, rotated rx 0 ry 90 rz 0 deg; joints [-9.348, 3.46, 52.635, 168.781, 56.606, -173.77]
  MoveL 1707 to (52.43, 41.12, 11) mm, rotated rx 0 ry 90 rz 0 deg; joints [-9.348, 3.417, 52.682, 168.781, 56.609, -173.77]
  Set speed (60.0 mm/s)
  Call Extruder(1064.653)
  MoveL 1708 to (58.01, 46.7, 11) mm, rotated rx 0 ry 90 rz 0 deg; joints [-9.639, 3.965, 51.178, 168.306, 55.704, -173.348]
  Call Extruder(1064.768)
  MoveL 1709 to (58.88, 46.7, 11) mm, rotated rx 0 ry 90 rz 0 deg; joints [-9.63, 4.039, 50.974, 168.299, 55.577, -173.323]
  Call Extruder(1065.510)
  MoveL 1710 to (58.88, 41.12, 11) mm, rotated rx 0 ry 90 rz 0 deg; joints [-9.282, 3.959, 51.193, 168.737, 55.673, -173.592]
  Call Extruder(1068.852)
  MoveL 1711 to (41.12, 58.88, 11) mm, rotated rx 0 ry 90 rz 0 deg; joints [-10.592, 2.763, 54.509, 167.468, 57.897, -173.263]
  Call Extruder(1068.852)
  MoveL 1712 to (41.12, 58.88, 11) mm, rotated rx 0 ry 90 rz 0 deg; joints [-10.592, 2.763, 54.509, 167.468, 57.897, -173.263]
  Call Extruder(1069.710)
  MoveL 1713 to (41.12, 52.43, 11) mm, rotated rx 0 ry 90 rz 0 deg; joints [-10.184, 2.671, 54.767, 167.967, 58.013, -173.558]
  Call Extruder(1070.923)
  MoveL 1714 to (47.57, 58.88, 11) mm, rotated rx 0 ry 90 rz 0 deg; joints [-10.516, 3.274, 53.08, 167.429, 56.992, -173.074]
  Call Extruder(1071.570)
  MoveL 1715 to (52.43, 58.88, 11) mm, rotated rx 0 ry 90 rz 0 deg; joints [-10.46, 3.674, 51.973, 167.395, 56.296, -172.926]
  Call Extruder(1072.778)
  MoveL 1716 to (58.85, 52.46, 11) mm, rotated rx 0 ry 90 rz 0 deg; joints [-9.988, 4.123, 50.746, 167.847, 55.478, -173.042]
  Call Extruder(1072.782)
  MoveL 1717 to (58.88, 52.46, 11) mm, rotated rx 0 ry 90 rz 0 deg; joints [-9.988, 4.126, 50.739, 167.847, 55.474, -173.041]
  Call Extruder(1073.636)
  MoveL 1718 to (58.88, 58.88, 11) mm, rotated rx 0 ry 90 rz 0 deg; joints [-10.386, 4.226, 50.466, 167.341, 55.354, -172.724]
  Call Extruder(1073.636)
  MoveL 1719 to (58.88, 58.88, 11) mm, rotated rx 0 ry 90 rz 0 deg; joints [-10.386, 4.226, 50.466, 167.342, 55.355, -172.724]
  Call Extruder(1076.978)
  MoveL 1720 to (41.12, 41.12, 11) mm, rotated rx 0 ry 90 rz 0 deg; joints [-9.467, 2.521, 55.192, 168.842, 58.205, -174.067]
  Call Extruder(1077.835)
  MoveL 1721 to (41.12, 47.56, 11) mm, rotated rx 0 ry 90 rz 0 deg; joints [-9.876, 2.605, 54.954, 168.344, 58.098, -173.778]
  Call Extruder(1078.951)
  MoveL 1722 to (47.05, 41.63, 11) mm, rotated rx 0 ry 90 rz 0 deg; joints [-9.437, 2.989, 53.873, 168.773, 57.367, -173.89]
  Call Extruder(1079.136)
  MoveL 1723 to (47.05, 43.02, 11) mm, rotated rx 0 ry 90 rz 0 deg; joints [-9.524, 3.008, 53.821, 168.666, 57.344, -173.827]
  Call Extruder(1079.784)
  MoveL 1724 to (51.93, 43.02, 11) mm, rotated rx 0 ry 90 rz 0 deg; joints [-9.473, 3.401, 52.726, 168.637, 56.65, -173.696]
  Call Extruder(1080.037)
  MoveL 1725 to (51.93, 41.12, 11) mm, rotated rx 0 ry 90 rz 0 deg; joints [-9.354, 3.376, 52.797, 168.785, 56.682, -173.784]
  Call Extruder(1080.962)
  MoveL 1726 to (58.88, 41.12, 11) mm, rotated rx 0 ry 90 rz 0 deg; joints [-9.282, 3.959, 51.193, 168.737, 55.673, -173.592]
  MoveL 1727 to (59.08, 41.12, 11) mm, rotated rx 0 ry 90 rz 0 deg; joints [-9.28, 3.976, 51.146, 168.735, 55.643, -173.587]
  Set speed (120.0 mm/s)
  MoveL 1728 to (51.23, 42.33, 11) mm, rotated rx 0 ry 90 rz 0 deg; joints [-9.437, 3.335, 52.909, 168.695, 56.761, -173.747]
  Set speed (1000.0 mm/s)
  MoveL 1729 to (47.7, 42.37, 11) mm, rotated rx 0 ry 90 rz 0 deg; joints [-9.476, 3.051, 53.701, 168.713, 57.263, -173.84]
  MoveL 1730 to (47.77, 42.3, 11) mm, rotated rx 0 ry 90 rz 0 deg; joints [-9.471, 3.056, 53.688, 168.718, 57.254, -173.841]
  Set speed (30.0 mm/s)
  Call Extruder(1081.015)
  MoveL 1731 to (48.17, 42.3, 11) mm, rotated rx 0 ry 90 rz 0 deg; joints [-9.467, 3.088, 53.599, 168.715, 57.198, -173.83]
  Call Extruder(1081.419)
  MoveL 1732 to (51.21, 42.3, 11) mm, rotated rx 0 ry 90 rz 0 deg; joints [-9.435, 3.333, 52.917, 168.697, 56.766, -173.749]
  Call Extruder(1081.671)
  MoveL 1733 to (51.21, 40.4, 11) mm, rotated rx 0 ry 90 rz 0 deg; joints [-9.316, 3.307, 52.987, 168.845, 56.797, -173.837]
  Call Extruder(1082.788)
  MoveL 1734 to (59.6, 40.4, 11) mm, rotated rx 0 ry 90 rz 0 deg; joints [-9.23, 4.011, 51.051, 168.788, 55.579, -173.606]
  Call Extruder(1083.722)
  MoveL 1735 to (59.6, 47.42, 11) mm, rotated rx 0 ry 90 rz 0 deg; joints [-9.667, 4.112, 50.776, 168.237, 55.458, -173.266]
  Call Extruder(1083.979)
  MoveL 1736 to (57.67, 47.42, 11) mm, rotated rx 0 ry 90 rz 0 deg; joints [-9.688, 3.945, 51.231, 168.252, 55.742, -173.323]
  Call Extruder(1084.553)
  MoveL 1737 to (57.66, 51.74, 11) mm, rotated rx 0 ry 90 rz 0 deg; joints [-9.956, 4.009, 51.056, 167.914, 55.666, -173.114]
  Call Extruder(1084.811)
  MoveL 1738 to (59.6, 51.74, 11) mm, rotated rx 0 ry 90 rz 0 deg; joints [-9.936, 4.177, 50.599, 167.897, 55.381, -173.054]
  Call Extruder(1085.857)
  MoveL 1739 to (59.6, 59.6, 11) mm, rotated rx 0 ry 90 rz 0 deg; joints [-10.423, 4.301, 50.263, 167.278, 55.234, -172.664]
  Call Extruder(1088.411)
  MoveL 1740 to (40.4, 59.6, 11) mm, rotated rx 0 ry 90 rz 0 deg; joints [-10.646, 2.718, 54.637, 167.416, 57.984, -173.25]
  Call Extruder(1090.965)
  MoveL 1741 to (40.4, 40.4, 11) mm, rotated rx 0 ry 90 rz 0 deg; joints [-9.429, 2.457, 55.374, 168.901, 58.317, -174.117]
  Call Extruder(1091.893)
  MoveL 1742 to (47.37, 40.4, 11) mm, rotated rx 0 ry 90 rz 0 deg; joints [-9.356, 2.999, 53.847, 168.867, 57.342, -173.938]
  Call Extruder(1091.946)
  MoveL 1743 to (47.77, 40.4, 11) mm, rotated rx 0 ry 90 rz 0 deg; joints [-9.351, 3.031, 53.758, 168.865, 57.285, -173.928]
  Call Extruder(1091.981)
  MoveL 1744 to (47.77, 40.8, 11) mm, rotated rx 0 ry 90 rz 0 deg; joints [-9.377, 3.036, 53.743, 168.834, 57.279, -173.91]
  Call Extruder(1092.127)
  MoveL 1745 to (47.77, 41.9, 11) mm, rotated rx 0 ry 90 rz 0 deg; joints [-9.446, 3.05, 53.703, 168.749, 57.261, -173.859]
  Call Extruder(1092.161)
  MoveL 1746 to (47.77, 42.3, 11) mm, rotated rx 0 ry 90 rz 0 deg; joints [-9.471, 3.056, 53.688, 168.718, 57.254, -173.841]
  Set speed (120.0 mm/s)
  MoveL 1747 to (48.17, 42.3, 11) mm, rotated rx 0 ry 90 rz 0 deg; joints [-9.467, 3.088, 53.599, 168.715, 57.198, -173.83]
  Set speed (1000.0 mm/s)
  MoveL 1748 to (48.17, 43.1, 11) mm, rotated rx 0 ry 90 rz 0 deg; joints [-9.518, 3.098, 53.569, 168.653, 57.184, -173.793]
  MoveL 1749 to (51.23, 42.33, 11) mm, rotated rx 0 ry 90 rz 0 deg; joints [-9.437, 3.335, 52.909, 168.695, 56.761, -173.747]
  MoveL 1750 to (52.43, 41.12, 11) mm, rotated rx 0 ry 90 rz 0 deg; joints [-9.348, 3.417, 52.682, 168.782, 56.609, -173.771]
  MoveL 1751 to (52.43, 41.12, 11.4) mm, rotated rx 0 ry 90 rz 0 deg; joints [-9.348, 3.374, 52.729, 168.782, 56.613, -173.771]
  Set speed (60.0 mm/s)
  Call Extruder(1093.166)
  MoveL 1752 to (57.77, 46.46, 11.4) mm, rotated rx 0 ry 90 rz 0 deg; joints [-9.627, 3.897, 51.291, 168.327, 55.747, -173.368]
  Call Extruder(1093.313)
  MoveL 1753 to (58.88, 46.46, 11.4) mm, rotated rx 0 ry 90 rz 0 deg; joints [-9.615, 3.992, 51.032, 168.319, 55.585, -173.335]
  Call Extruder(1094.024)
  MoveL 1754 to (58.88, 41.12, 11.4) mm, rotated rx 0 ry 90 rz 0 deg; joints [-9.282, 3.916, 51.241, 168.737, 55.677, -173.593]
  Call Extruder(1097.366)
  MoveL 1755 to (41.12, 58.88, 11.4) mm, rotated rx 0 ry 90 rz 0 deg; joints [-10.592, 2.72, 54.554, 167.468, 57.9, -173.263]
  Call Extruder(1097.366)
  MoveL 1756 to (41.12, 58.88, 11.4) mm, rotated rx 0 ry 90 rz 0 deg; joints [-10.592, 2.72, 54.554, 167.468, 57.9, -173.263]
  Call Extruder(1098.224)
  MoveL 1757 to (41.12, 52.43, 11.4) mm, rotated rx 0 ry 90 rz 0 deg; joints [-10.184, 2.629, 54.812, 167.968, 58.016, -173.559]
  Call Extruder(1099.436)
  MoveL 1758 to (47.56, 58.88, 11.4) mm, rotated rx 0 ry 90 rz 0 deg; joints [-10.516, 3.231, 53.126, 167.43, 56.995, -173.075]
  Call Extruder(1100.084)
  MoveL 1759 to (52.43, 58.88, 11.4) mm, rotated rx 0 ry 90 rz 0 deg; joints [-10.46, 3.631, 52.02, 167.395, 56.299, -172.927]
  Call Extruder(1101.250)
  MoveL 1760 to (58.63, 52.68, 11.4) mm, rotated rx 0 ry 90 rz 0 deg; joints [-10.005, 4.064, 50.837, 167.832, 55.511, -173.039]
  Call Extruder(1101.283)
  MoveL 1761 to (58.88, 52.68, 11.4) mm, rotated rx 0 ry 90 rz 0 deg; joints [-10.002, 4.086, 50.778, 167.83, 55.474, -173.031]
  Call Extruder(1102.107)
  MoveL 1762 to (58.88, 58.88, 11.4) mm, rotated rx 0 ry 90 rz 0 deg; joints [-10.386, 4.183, 50.514, 167.342, 55.359, -172.725]
  Call Extruder(1102.107)
  MoveL 1763 to (58.88, 58.88, 11.4) mm, rotated rx 0 ry 90 rz 0 deg; joints [-10.386, 4.183, 50.514, 167.342, 55.359, -172.725]
  Call Extruder(1105.449)
  MoveL 1764 to (41.12, 41.12, 11.4) mm, rotated rx 0 ry 90 rz 0 deg; joints [-9.467, 2.479, 55.237, 168.842, 58.208, -174.067]
  Call Extruder(1106.307)
  MoveL 1765 to (41.12, 47.56, 11.4) mm, rotated rx 0 ry 90 rz 0 deg; joints [-9.876, 2.563, 54.999, 168.344, 58.1, -173.779]
  Call Extruder(1107.380)
  MoveL 1766 to (46.83, 41.86, 11.4) mm, rotated rx 0 ry 90 rz 0 deg; joints [-9.453, 2.932, 53.96, 168.757, 57.398, -173.887]
  Call Extruder(1107.535)
  MoveL 1767 to (46.83, 43.02, 11.4) mm, rotated rx 0 ry 90 rz 0 deg; joints [-9.527, 2.947, 53.917, 168.667, 57.379, -173.834]
  Call Extruder(1108.247)
  MoveL 1768 to (52.18, 43.02, 11.4) mm, rotated rx 0 ry 90 rz 0 deg; joints [-9.47, 3.379, 52.715, 168.636, 56.617, -173.689]
  Call Extruder(1108.500)
  MoveL 1769 to (52.18, 41.12, 11.4) mm, rotated rx 0 ry 90 rz 0 deg; joints [-9.351, 3.354, 52.786, 168.783, 56.649, -173.778]
  Call Extruder(1109.391)
  MoveL 1770 to (58.88, 41.12, 11.4) mm, rotated rx 0 ry 90 rz 0 deg; joints [-9.282, 3.916, 51.24, 168.737, 55.677, -173.593]
  MoveL 1771 to (59.08, 41.12, 11.4) mm, rotated rx 0 ry 90 rz 0 deg; joints [-9.28, 3.933, 51.193, 168.736, 55.647, -173.588]
  Set speed (120.0 mm/s)
  MoveL 1772 to (51.49, 42.33, 11.4) mm, rotated rx 0 ry 90 rz 0 deg; joints [-9.434, 3.313, 52.898, 168.694, 56.728, -173.741]
  Set speed (1000.0 mm/s)
  MoveL 1773 to (47.48, 42.37, 11.4) mm, rotated rx 0 ry 90 rz 0 deg; joints [-9.479, 2.99, 53.797, 168.714, 57.298, -173.846]
  MoveL 1774 to (47.55, 42.3, 11.4) mm, rotated rx 0 ry 90 rz 0 deg; joints [-9.474, 2.995, 53.784, 168.719, 57.289, -173.848]
  Set speed (30.0 mm/s)
  Call Extruder(1109.444)
  MoveL 1775 to (47.95, 42.3, 11.4) mm, rotated rx 0 ry 90 rz 0 deg; joints [-9.469, 3.027, 53.695, 168.717, 57.232, -173.837]
  Call Extruder(1109.912)
  MoveL 1776 to (51.46, 42.3, 11.4) mm, rotated rx 0 ry 90 rz 0 deg; joints [-9.433, 3.311, 52.905, 168.696, 56.732, -173.743]
  Call Extruder(1110.164)
  MoveL 1777 to (51.46, 40.4, 11.4) mm, rotated rx 0 ry 90 rz 0 deg; joints [-9.313, 3.285, 52.976, 168.844, 56.764, -173.831]
  Call Extruder(1111.247)
  MoveL 1778 to (59.6, 40.4, 11.4) mm, rotated rx 0 ry 90 rz 0 deg; joints [-9.23, 3.968, 51.099, 168.788, 55.583, -173.607]
  Call Extruder(1112.149)
  MoveL 1779 to (59.6, 47.18, 11.4) mm, rotated rx 0 ry 90 rz 0 deg; joints [-9.652, 4.065, 50.833, 168.257, 55.466, -173.279]
  Call Extruder(1112.406)
  MoveL 1780 to (57.67, 47.18, 11.4) mm, rotated rx 0 ry 90 rz 0 deg; joints [-9.673, 3.899, 51.287, 168.272, 55.75, -173.336]
  Call Extruder(1112.714)
  MoveL 1781 to (57.67, 49.49, 11.4) mm, rotated rx 0 ry 90 rz 0 deg; joints [-9.817, 3.933, 51.194, 168.091, 55.71, -173.224]
  Call Extruder(1113.042)
  MoveL 1782 to (57.67, 51.96, 11.4) mm, rotated rx 0 ry 90 rz 0 deg; joints [-9.97, 3.969, 51.094, 167.897, 55.666, -173.104]
  Call Extruder(1113.300)
  MoveL 1783 to (59.6, 51.97, 11.4) mm, rotated rx 0 ry 90 rz 0 deg; joints [-9.95, 4.137, 50.637, 167.88, 55.381, -173.044]
  Call Extruder(1114.315)
  MoveL 1784 to (59.6, 59.6, 11.4) mm, rotated rx 0 ry 90 rz 0 deg; joints [-10.423, 4.257, 50.311, 167.279, 55.239, -172.666]
  Call Extruder(1116.869)
  MoveL 1785 to (40.4, 59.6, 11.4) mm, rotated rx 0 ry 90 rz 0 deg; joints [-10.646, 2.675, 54.682, 167.416, 57.986, -173.251]
  Call Extruder(1119.424)
  MoveL 1786 to (40.4, 40.4, 11.4) mm, rotated rx 0 ry 90 rz 0 deg; joints [-9.429, 2.415, 55.418, 168.901, 58.319, -174.118]
  Call Extruder(1120.322)
  MoveL 1787 to (47.15, 40.4, 11.4) mm, rotated rx 0 ry 90 rz 0 deg; joints [-9.358, 2.938, 53.942, 168.869, 57.377, -173.945]
  Call Extruder(1120.375)
  MoveL 1788 to (47.55, 40.4, 11.4) mm, rotated rx 0 ry 90 rz 0 deg; joints [-9.354, 2.97, 53.854, 168.866, 57.32, -173.934]
  Call Extruder(1120.409)
  MoveL 1789 to (47.55, 40.8, 11.4) mm, rotated rx 0 ry 90 rz 0 deg; joints [-9.379, 2.975, 53.839, 168.835, 57.314, -173.916]
  Call Extruder(1120.555)
  MoveL 1790 to (47.55, 41.9, 11.4) mm, rotated rx 0 ry 90 rz 0 deg; joints [-9.448, 2.99, 53.799, 168.75, 57.296, -173.866]
  Call Extruder(1120.590)
  MoveL 1791 to (47.55, 42.3, 11.4) mm, rotated rx 0 ry 90 rz 0 deg; joints [-9.474, 2.995, 53.784, 168.719, 57.289, -173.848]
  Set speed (120.0 mm/s)
  MoveL 1792 to (47.95, 42.3, 11.4) mm, rotated rx 0 ry 90 rz 0 deg; joints [-9.469, 3.027, 53.695, 168.717, 57.232, -173.837]
  Set speed (1000.0 mm/s)
  MoveL 1793 to (47.95, 43.1, 11.4) mm, rotated rx 0 ry 90 rz 0 deg; joints [-9.52, 3.037, 53.665, 168.655, 57.219, -173.8]
  MoveL 1794 to (51.49, 42.33, 11.4) mm, rotated rx 0 ry 90 rz 0 deg; joints [-9.434, 3.313, 52.898, 168.694, 56.728, -173.741]
  MoveL 1795 to (52.44, 41.12, 11.4) mm, rotated rx 0 ry 90 rz 0 deg; joints [-9.349, 3.374, 52.728, 168.782, 56.612, -173.771]
  MoveL 1796 to (52.43, 41.12, 11.8) mm, rotated rx 0 ry 90 rz 0 deg; joints [-9.349, 3.331, 52.775, 168.782, 56.616, -173.772]
  Set speed (60.0 mm/s)
  Call Extruder(1121.550)
  MoveL 1797 to (57.54, 46.22, 11.8) mm, rotated rx 0 ry 90 rz 0 deg; joints [-9.614, 3.83, 51.404, 168.349, 55.79, -173.387]
  Call Extruder(1121.728)
  MoveL 1798 to (58.88, 46.22, 11.8) mm, rotated rx 0 ry 90 rz 0 deg; joints [-9.6, 3.945, 51.089, 168.338, 55.593, -173.348]
  Call Extruder(1122.407)
  MoveL 1799 to (58.88, 41.12, 11.8) mm, rotated rx 0 ry 90 rz 0 deg; joints [-9.282, 3.872, 51.288, 168.738, 55.681, -173.594]
  Call Extruder(1125.749)
  MoveL 1800 to (41.12, 58.88, 11.8) mm, rotated rx 0 ry 90 rz 0 deg; joints [-10.592, 2.678, 54.6, 167.468, 57.903, -173.264]
  Call Extruder(1125.749)
  MoveL 1801 to (41.12, 58.88, 11.8) mm, rotated rx 0 ry 90 rz 0 deg; joints [-10.592, 2.678, 54.599, 167.468, 57.902, -173.264]
  Call Extruder(1126.607)
  MoveL 1802 to (41.12, 52.43, 11.8) mm, rotated rx 0 ry 90 rz 0 deg; joints [-10.184, 2.587, 54.857, 167.968, 58.018, -173.559]
  Call Extruder(1127.820)
  MoveL 1803 to (47.56, 58.88, 11.8) mm, rotated rx 0 ry 90 rz 0 deg; joints [-10.516, 3.188, 53.172, 167.43, 56.998, -173.076]
  Call Extruder(1128.467)
  MoveL 1804 to (52.43, 58.88, 11.8) mm, rotated rx 0 ry 90 rz 0 deg; joints [-10.46, 3.588, 52.067, 167.396, 56.303, -172.928]
  Call Extruder(1129.590)
  MoveL 1805 to (58.4, 52.91, 11.8) mm, rotated rx 0 ry 90 rz 0 deg; joints [-10.021, 4.004, 50.929, 167.817, 55.544, -173.036]
  Call Extruder(1129.654)
  MoveL 1806 to (58.88, 52.91, 11.8) mm, rotated rx 0 ry 90 rz 0 deg; joints [-10.016, 4.045, 50.816, 167.813, 55.474, -173.021]
  Call Extruder(1130.448)
  MoveL 1807 to (58.88, 58.88, 11.8) mm, rotated rx 0 ry 90 rz 0 deg; joints [-10.386, 4.139, 50.562, 167.343, 55.363, -172.726]
  Call Extruder(1130.448)
  MoveL 1808 to (58.88, 58.88, 11.8) mm, rotated rx 0 ry 90 rz 0 deg; joints [-10.386, 4.139, 50.562, 167.343, 55.363, -172.726]
  Call Extruder(1133.790)
  MoveL 1809 to (41.12, 41.12, 11.8) mm, rotated rx 0 ry 90 rz 0 deg; joints [-9.467, 2.436, 55.282, 168.843, 58.21, -174.068]
  Call Extruder(1134.647)
  MoveL 1810 to (41.12, 47.57, 11.8) mm, rotated rx 0 ry 90 rz 0 deg; joints [-9.876, 2.52, 55.044, 168.345, 58.102, -173.779]
  Call Extruder(1135.678)
  MoveL 1811 to (46.6, 42.08, 11.8) mm, rotated rx 0 ry 90 rz 0 deg; joints [-9.47, 2.874, 54.047, 168.741, 57.429, -173.883]
  Call Extruder(1135.803)
  MoveL 1812 to (46.6, 43.02, 11.8) mm, rotated rx 0 ry 90 rz 0 deg; joints [-9.529, 2.887, 54.013, 168.669, 57.413, -173.84]
  Call Extruder(1136.579)
  MoveL 1813 to (52.44, 43.02, 11.8) mm, rotated rx 0 ry 90 rz 0 deg; joints [-9.468, 3.357, 52.703, 168.635, 56.584, -173.683]
  Call Extruder(1136.832)
  MoveL 1814 to (52.44, 41.12, 11.8) mm, rotated rx 0 ry 90 rz 0 deg; joints [-9.348, 3.332, 52.774, 168.782, 56.616, -173.772]
  Call Extruder(1137.689)
  MoveL 1815 to (58.88, 41.12, 11.8) mm, rotated rx 0 ry 90 rz 0 deg; joints [-9.282, 3.872, 51.288, 168.738, 55.681, -173.594]
  MoveL 1816 to (59.08, 41.12, 11.8) mm, rotated rx 0 ry 90 rz 0 deg; joints [-9.28, 3.89, 51.241, 168.736, 55.651, -173.588]
  Set speed (120.0 mm/s)
  MoveL 1817 to (57.64, 46.92, 11.8) mm, rotated rx 0 ry 90 rz 0 deg; joints [-9.656, 3.849, 51.352, 168.293, 55.763, -173.351]
  Set speed (1000.0 mm/s)
  MoveL 1818 to (57.6, 49.5, 11.8) mm, rotated rx 0 ry 90 rz 0 deg; joints [-9.818, 3.883, 51.258, 168.091, 55.724, -173.227]
  MoveL 1819 to (57.67, 49.43, 11.8) mm, rotated rx 0 ry 90 rz 0 deg; joints [-9.813, 3.888, 51.244, 168.096, 55.715, -173.228]
  Set speed (30.0 mm/s)
  Call Extruder(1137.742)
  MoveL 1820 to (58.07, 49.43, 11.8) mm, rotated rx 0 ry 90 rz 0 deg; joints [-9.808, 3.923, 51.151, 168.093, 55.656, -173.216]
  Call Extruder(1137.946)
  MoveL 1821 to (59.6, 49.43, 11.8) mm, rotated rx 0 ry 90 rz 0 deg; joints [-9.792, 4.055, 50.79, 168.081, 55.431, -173.17]
  Call Extruder(1137.985)
  MoveL 1822 to (59.6, 49.72, 11.8) mm, rotated rx 0 ry 90 rz 0 deg; joints [-9.81, 4.06, 50.778, 168.058, 55.426, -173.156]
  Call Extruder(1138.189)
  MoveL 1823 to (58.07, 49.72, 11.8) mm, rotated rx 0 ry 90 rz 0 deg; joints [-9.826, 3.927, 51.139, 168.07, 55.651, -173.202]
  Call Extruder(1138.243)
  MoveL 1824 to (57.67, 49.72, 11.8) mm, rotated rx 0 ry 90 rz 0 deg; joints [-9.831, 3.892, 51.233, 168.074, 55.71, -173.214]
  Call Extruder(1138.277)
  MoveL 1825 to (57.67, 50.12, 11.8) mm, rotated rx 0 ry 90 rz 0 deg; joints [-9.856, 3.898, 51.217, 168.042, 55.703, -173.195]
  Call Extruder(1138.553)
  MoveL 1826 to (57.67, 52.19, 11.8) mm, rotated rx 0 ry 90 rz 0 deg; joints [-9.985, 3.929, 51.132, 167.88, 55.666, -173.094]
  Call Extruder(1138.810)
  MoveL 1827 to (59.6, 52.19, 11.8) mm, rotated rx 0 ry 90 rz 0 deg; joints [-9.964, 4.097, 50.676, 167.863, 55.381, -173.034]
  Call Extruder(1139.795)
  MoveL 1828 to (59.6, 59.6, 11.8) mm, rotated rx 0 ry 90 rz 0 deg; joints [-10.423, 4.214, 50.36, 167.279, 55.243, -172.667]
  Call Extruder(1142.350)
  MoveL 1829 to (40.4, 59.6, 11.8) mm, rotated rx 0 ry 90 rz 0 deg; joints [-10.646, 2.633, 54.727, 167.416, 57.989, -173.252]
  Call Extruder(1144.904)
  MoveL 1830 to (40.4, 40.4, 11.8) mm, rotated rx 0 ry 90 rz 0 deg; joints [-9.429, 2.373, 55.463, 168.901, 58.321, -174.118]
  Call Extruder(1145.772)
  MoveL 1831 to (46.92, 40.4, 11.8) mm, rotated rx 0 ry 90 rz 0 deg; joints [-9.36, 2.878, 54.038, 168.87, 57.411, -173.951]
  Call Extruder(1145.825)
  MoveL 1832 to (47.32, 40.4, 11.8) mm, rotated rx 0 ry 90 rz 0 deg; joints [-9.356, 2.909, 53.949, 168.868, 57.355, -173.941]
  Call Extruder(1145.860)
  MoveL 1833 to (47.32, 40.8, 11.8) mm, rotated rx 0 ry 90 rz 0 deg; joints [-9.381, 2.915, 53.935, 168.837, 57.348, -173.923]
  Call Extruder(1146.006)
  MoveL 1834 to (47.32, 41.9, 11.8) mm, rotated rx 0 ry 90 rz 0 deg; joints [-9.451, 2.929, 53.894, 168.752, 57.33, -173.873]
  Call Extruder(1146.059)
  MoveL 1835 to (47.32, 42.3, 11.8) mm, rotated rx 0 ry 90 rz 0 deg; joints [-9.476, 2.934, 53.879, 168.721, 57.324, -173.854]
  Call Extruder(1146.093)
  MoveL 1836 to (47.72, 42.3, 11.8) mm, rotated rx 0 ry 90 rz 0 deg; joints [-9.472, 2.966, 53.791, 168.719, 57.267, -173.844]
  Call Extruder(1146.572)
  MoveL 1837 to (51.32, 42.3, 11.8) mm, rotated rx 0 ry 90 rz 0 deg; joints [-9.434, 3.256, 52.984, 168.698, 56.756, -173.747]
  Call Extruder(1146.625)
  MoveL 1838 to (51.72, 42.3, 11.8) mm, rotated rx 0 ry 90 rz 0 deg; joints [-9.43, 3.289, 52.893, 168.695, 56.699, -173.736]
  Call Extruder(1146.659)
  MoveL 1839 to (51.72, 41.9, 11.8) mm, rotated rx 0 ry 90 rz 0 deg; joints [-9.405, 3.283, 52.908, 168.726, 56.706, -173.755]
  Call Extruder(1146.805)
  MoveL 1840 to (51.72, 40.8, 11.8) mm, rotated rx 0 ry 90 rz 0 deg; joints [-9.336, 3.268, 52.95, 168.812, 56.724, -173.806]
  Call Extruder(1146.859)
  MoveL 1841 to (51.72, 40.4, 11.8) mm, rotated rx 0 ry 90 rz 0 deg; joints [-9.311, 3.263, 52.965, 168.843, 56.731, -173.825]
  Call Extruder(1146.893)
  MoveL 1842 to (52.12, 40.4, 11.8) mm, rotated rx 0 ry 90 rz 0 deg; joints [-9.307, 3.296, 52.874, 168.84, 56.674, -173.814]
  Call Extruder(1147.889)
  MoveL 1843 to (59.6, 40.4, 11.8) mm, rotated rx 0 ry 90 rz 0 deg; joints [-9.23, 3.924, 51.146, 168.789, 55.587, -173.608]
  Call Extruder(1148.759)
  MoveL 1844 to (59.6, 46.94, 11.8) mm, rotated rx 0 ry 90 rz 0 deg; joints [-9.637, 4.018, 50.89, 168.276, 55.475, -173.292]
  Call Extruder(1149.016)
  MoveL 1845 to (57.67, 46.94, 11.8) mm, rotated rx 0 ry 90 rz 0 deg; joints [-9.658, 3.852, 51.344, 168.291, 55.759, -173.348]
  Call Extruder(1149.293)
  MoveL 1846 to (57.67, 49.03, 11.8) mm, rotated rx 0 ry 90 rz 0 deg; joints [-9.788, 3.882, 51.261, 168.128, 55.722, -173.247]
  Call Extruder(1149.328)
  MoveL 1847 to (57.67, 49.43, 11.8) mm, rotated rx 0 ry 90 rz 0 deg; joints [-9.813, 3.888, 51.244, 168.096, 55.715, -173.228]
  Set speed (120.0 mm/s)
  MoveL 1848 to (58.07, 49.43, 11.8) mm, rotated rx 0 ry 90 rz 0 deg; joints [-9.808, 3.923, 51.151, 168.093, 55.656, -173.216]
  Set speed (1000.0 mm/s)
  MoveL 1849 to (56.87, 50.23, 11.8) mm, rotated rx 0 ry 90 rz 0 deg; joints [-9.871, 3.832, 51.4, 168.04, 55.818, -173.213]
  MoveL 1850 to (52.69, 41.38, 11.8) mm, rotated rx 0 ry 90 rz 0 deg; joints [-9.362, 3.356, 52.707, 168.761, 56.575, -173.753]
  MoveL 1851 to (52.69, 41.38, 12.2) mm, rotated rx 0 ry 90 rz 0 deg; joints [-9.362, 3.313, 52.753, 168.761, 56.578, -173.754]
  Set speed (60.0 mm/s)
  Call Extruder(1150.194)
  MoveL 1852 to (57.3, 45.98, 12.2) mm, rotated rx 0 ry 90 rz 0 deg; joints [-9.602, 3.763, 51.516, 168.37, 55.833, -173.406]
  Call Extruder(1150.405)
  MoveL 1853 to (58.88, 45.98, 12.2) mm, rotated rx 0 ry 90 rz 0 deg; joints [-9.585, 3.898, 51.146, 168.357, 55.602, -173.36]
  Call Extruder(1151.052)
  MoveL 1854 to (58.88, 41.12, 12.2) mm, rotated rx 0 ry 90 rz 0 deg; joints [-9.282, 3.829, 51.335, 168.738, 55.685, -173.595]
  Call Extruder(1154.394)
  MoveL 1855 to (41.12, 58.88, 12.2) mm, rotated rx 0 ry 90 rz 0 deg; joints [-10.592, 2.635, 54.645, 167.469, 57.905, -173.265]
  Call Extruder(1154.394)
  MoveL 1856 to (41.12, 58.88, 12.2) mm, rotated rx 0 ry 90 rz 0 deg; joints [-10.592, 2.636, 54.644, 167.469, 57.905, -173.265]
  Call Extruder(1155.251)
  MoveL 1857 to (41.12, 52.43, 12.2) mm, rotated rx 0 ry 90 rz 0 deg; joints [-10.184, 2.544, 54.902, 167.968, 58.021, -173.56]
  Call Extruder(1156.464)
  MoveL 1858 to (47.56, 58.88, 12.2) mm, rotated rx 0 ry 90 rz 0 deg; joints [-10.516, 3.145, 53.218, 167.431, 57.002, -173.076]
  Call Extruder(1157.112)
  MoveL 1859 to (52.43, 58.88, 12.2) mm, rotated rx 0 ry 90 rz 0 deg; joints [-10.46, 3.545, 52.113, 167.397, 56.306, -172.929]
  Call Extruder(1158.192)
  MoveL 1860 to (58.17, 53.14, 12.2) mm, rotated rx 0 ry 90 rz 0 deg; joints [-10.038, 3.944, 51.021, 167.801, 55.578, -173.033]
  Call Extruder(1158.286)
  MoveL 1861 to (58.88, 53.14, 12.2) mm, rotated rx 0 ry 90 rz 0 deg; joints [-10.03, 4.005, 50.854, 167.795, 55.474, -173.011]
  Call Extruder(1159.050)
  MoveL 1862 to (58.88, 58.88, 12.2) mm, rotated rx 0 ry 90 rz 0 deg; joints [-10.386, 4.095, 50.61, 167.343, 55.367, -172.727]
  Call Extruder(1159.050)
  MoveL 1863 to (58.88, 58.88, 12.2) mm, rotated rx 0 ry 90 rz 0 deg; joints [-10.386, 4.095, 50.61, 167.344, 55.368, -172.727]
  Call Extruder(1162.391)
  MoveL 1864 to (41.12, 41.12, 12.2) mm, rotated rx 0 ry 90 rz 0 deg; joints [-9.467, 2.394, 55.327, 168.843, 58.212, -174.069]
  Call Extruder(1163.249)
  MoveL 1865 to (41.12, 47.57, 12.2) mm, rotated rx 0 ry 90 rz 0 deg; joints [-9.876, 2.478, 55.089, 168.345, 58.105, -173.78]
  Call Extruder(1164.238)
  MoveL 1866 to (46.38, 42.31, 12.2) mm, rotated rx 0 ry 90 rz 0 deg; joints [-9.487, 2.817, 54.134, 168.725, 57.46, -173.879]
  Call Extruder(1164.332)
  MoveL 1867 to (46.38, 43.02, 12.2) mm, rotated rx 0 ry 90 rz 0 deg; joints [-9.532, 2.827, 54.108, 168.67, 57.448, -173.847]
  Call Extruder(1165.173)
  MoveL 1868 to (52.69, 43.02, 12.2) mm, rotated rx 0 ry 90 rz 0 deg; joints [-9.465, 3.336, 52.691, 168.633, 56.55, -173.677]
  Call Extruder(1165.426)
  MoveL 1869 to (52.69, 41.12, 12.2) mm, rotated rx 0 ry 90 rz 0 deg; joints [-9.346, 3.31, 52.763, 168.781, 56.582, -173.766]
  Call Extruder(1166.249)
  MoveL 1870 to (58.88, 41.12, 12.2) mm, rotated rx 0 ry 90 rz 0 deg; joints [-9.282, 3.829, 51.335, 168.738, 55.685, -173.595]
  MoveL 1871 to (59.08, 41.12, 12.2) mm, rotated rx 0 ry 90 rz 0 deg; joints [-9.28, 3.846, 51.288, 168.737, 55.655, -173.589]
  Set speed (120.0 mm/s)
  MoveL 1872 to (57.64, 46.68, 12.2) mm, rotated rx 0 ry 90 rz 0 deg; joints [-9.642, 3.802, 51.409, 168.313, 55.771, -173.363]
  Set speed (1000.0 mm/s)
  MoveL 1873 to (57.6, 49.87, 12.2) mm, rotated rx 0 ry 90 rz 0 deg; joints [-9.841, 3.845, 51.291, 168.063, 55.721, -173.21]
  MoveL 1874 to (57.67, 49.94, 12.2) mm, rotated rx 0 ry 90 rz 0 deg; joints [-9.844, 3.852, 51.271, 168.057, 55.71, -173.204]
  Set speed (30.0 mm/s)
  Call Extruder(1166.302)
  MoveL 1875 to (57.67, 50.34, 12.2) mm, rotated rx 0 ry 90 rz 0 deg; joints [-9.869, 3.858, 51.255, 168.025, 55.703, -173.185]
  Call Extruder(1166.579)
  MoveL 1876 to (57.67, 52.42, 12.2) mm, rotated rx 0 ry 90 rz 0 deg; joints [-9.999, 3.89, 51.17, 167.862, 55.665, -173.084]
  Call Extruder(1166.836)
  MoveL 1877 to (59.6, 52.42, 12.2) mm, rotated rx 0 ry 90 rz 0 deg; joints [-9.978, 4.057, 50.714, 167.846, 55.381, -173.024]
  Call Extruder(1167.791)
  MoveL 1878 to (59.6, 59.6, 12.2) mm, rotated rx 0 ry 90 rz 0 deg; joints [-10.423, 4.17, 50.408, 167.28, 55.248, -172.668]
  Call Extruder(1170.345)
  MoveL 1879 to (40.4, 59.6, 12.2) mm, rotated rx 0 ry 90 rz 0 deg; joints [-10.646, 2.59, 54.772, 167.417, 57.992, -173.252]
  Call Extruder(1172.900)
  MoveL 1880 to (40.4, 40.4, 12.2) mm, rotated rx 0 ry 90 rz 0 deg; joints [-9.429, 2.33, 55.508, 168.901, 58.323, -174.119]
  Call Extruder(1173.738)
  MoveL 1881 to (46.7, 40.4, 12.2) mm, rotated rx 0 ry 90 rz 0 deg; joints [-9.363, 2.817, 54.133, 168.872, 57.446, -173.958]
  Call Extruder(1173.791)
  MoveL 1882 to (47.1, 40.4, 12.2) mm, rotated rx 0 ry 90 rz 0 deg; joints [-9.358, 2.849, 54.045, 168.87, 57.39, -173.948]
  Call Extruder(1173.825)
  MoveL 1883 to (47.1, 40.8, 12.2) mm, rotated rx 0 ry 90 rz 0 deg; joints [-9.384, 2.854, 54.03, 168.839, 57.383, -173.929]
  Call Extruder(1173.972)
  MoveL 1884 to (47.1, 41.9, 12.2) mm, rotated rx 0 ry 90 rz 0 deg; joints [-9.453, 2.869, 53.99, 168.753, 57.365, -173.879]
  Call Extruder(1174.025)
  MoveL 1885 to (47.1, 42.3, 12.2) mm, rotated rx 0 ry 90 rz 0 deg; joints [-9.478, 2.874, 53.975, 168.722, 57.358, -173.861]
  Call Extruder(1174.059)
  MoveL 1886 to (47.5, 42.3, 12.2) mm, rotated rx 0 ry 90 rz 0 deg; joints [-9.474, 2.906, 53.886, 168.72, 57.302, -173.85]
  Call Extruder(1174.602)
  MoveL 1887 to (51.57, 42.3, 12.2) mm, rotated rx 0 ry 90 rz 0 deg; joints [-9.431, 3.234, 52.972, 168.696, 56.723, -173.741]
  Call Extruder(1174.655)
  MoveL 1888 to (51.97, 42.3, 12.2) mm, rotated rx 0 ry 90 rz 0 deg; joints [-9.427, 3.267, 52.882, 168.694, 56.666, -173.73]
  Call Extruder(1174.689)
  MoveL 1889 to (51.97, 41.9, 12.2) mm, rotated rx 0 ry 90 rz 0 deg; joints [-9.402, 3.261, 52.897, 168.725, 56.672, -173.749]
  Call Extruder(1174.835)
  MoveL 1890 to (51.97, 40.8, 12.2) mm, rotated rx 0 ry 90 rz 0 deg; joints [-9.333, 3.246, 52.938, 168.811, 56.691, -173.8]
  Call Extruder(1174.889)
  MoveL 1891 to (51.97, 40.4, 12.2) mm, rotated rx 0 ry 90 rz 0 deg; joints [-9.308, 3.241, 52.953, 168.842, 56.698, -173.819]
  Call Extruder(1174.923)
  MoveL 1892 to (52.37, 40.4, 12.2) mm, rotated rx 0 ry 90 rz 0 deg; joints [-9.304, 3.274, 52.862, 168.839, 56.64, -173.808]
  Call Extruder(1175.885)
  MoveL 1893 to (59.6, 40.4, 12.2) mm, rotated rx 0 ry 90 rz 0 deg; joints [-9.23, 3.881, 51.194, 168.789, 55.591, -173.609]
  Call Extruder(1176.723)
  MoveL 1894 to (59.6, 46.7, 12.2) mm, rotated rx 0 ry 90 rz 0 deg; joints [-9.622, 3.971, 50.948, 168.295, 55.483, -173.304]
  Call Extruder(1176.980)
  MoveL 1895 to (57.67, 46.7, 12.2) mm, rotated rx 0 ry 90 rz 0 deg; joints [-9.643, 3.805, 51.401, 168.31, 55.767, -173.361]
  Call Extruder(1177.258)
  MoveL 1896 to (57.67, 48.79, 12.2) mm, rotated rx 0 ry 90 rz 0 deg; joints [-9.773, 3.836, 51.317, 168.147, 55.73, -173.26]
  Call Extruder(1177.311)
  MoveL 1897 to (57.67, 49.19, 12.2) mm, rotated rx 0 ry 90 rz 0 deg; joints [-9.798, 3.841, 51.301, 168.115, 55.723, -173.24]
  Call Extruder(1177.346)
  MoveL 1898 to (58.07, 49.19, 12.2) mm, rotated rx 0 ry 90 rz 0 deg; joints [-9.794, 3.876, 51.208, 168.112, 55.664, -173.229]
  Call Extruder(1177.550)
  MoveL 1899 to (59.6, 49.19, 12.2) mm, rotated rx 0 ry 90 rz 0 deg; joints [-9.777, 4.008, 50.847, 168.1, 55.439, -173.183]
  Call Extruder(1177.650)
  MoveL 1900 to (59.6, 49.94, 12.2) mm, rotated rx 0 ry 90 rz 0 deg; joints [-9.824, 4.019, 50.817, 168.041, 55.426, -173.146]
  Call Extruder(1177.847)
  MoveL 1901 to (58.07, 49.94, 12.2) mm, rotated rx 0 ry 90 rz 0 deg; joints [-9.84, 3.887, 51.178, 168.054, 55.651, -173.192]
  Call Extruder(1177.882)
  MoveL 1902 to (57.67, 49.94, 12.2) mm, rotated rx 0 ry 90 rz 0 deg; joints [-9.844, 3.852, 51.271, 168.057, 55.71, -173.204]
  Set speed (120.0 mm/s)
  MoveL 1903 to (57.67, 50.34, 12.2) mm, rotated rx 0 ry 90 rz 0 deg; joints [-9.869, 3.858, 51.255, 168.025, 55.703, -173.185]
  Set speed (1000.0 mm/s)
  MoveL 1904 to (56.87, 50.34, 12.2) mm, rotated rx 0 ry 90 rz 0 deg; joints [-9.878, 3.79, 51.442, 168.032, 55.82, -173.209]
  MoveL 1905 to (52.95, 41.63, 12.2) mm, rotated rx 0 ry 90 rz 0 deg; joints [-9.375, 3.337, 52.686, 168.74, 56.537, -173.735]
  MoveL 1906 to (52.95, 41.63, 12.6) mm, rotated rx 0 ry 90 rz 0 deg; joints [-9.375, 3.295, 52.732, 168.74, 56.541, -173.736]
  Set speed (60.0 mm/s)
  Call Extruder(1178.656)
  MoveL 1907 to (57.06, 45.75, 12.6) mm, rotated rx 0 ry 90 rz 0 deg; joints [-9.59, 3.696, 51.628, 168.391, 55.876, -173.426]
  Call Extruder(1178.898)
  MoveL 1908 to (58.88, 45.74, 12.6) mm, rotated rx 0 ry 90 rz 0 deg; joints [-9.57, 3.852, 51.203, 168.377, 55.61, -173.373]
  Call Extruder(1179.513)
  MoveL 1909 to (58.88, 41.12, 12.6) mm, rotated rx 0 ry 90 rz 0 deg; joints [-9.282, 3.786, 51.383, 168.739, 55.689, -173.596]
  Call Extruder(1182.855)
  MoveL 1910 to (41.12, 58.88, 12.6) mm, rotated rx 0 ry 90 rz 0 deg; joints [-10.592, 2.593, 54.69, 167.469, 57.908, -173.266]
  Call Extruder(1182.855)
  MoveL 1911 to (41.12, 58.88, 12.6) mm, rotated rx 0 ry 90 rz 0 deg; joints [-10.592, 2.593, 54.689, 167.469, 57.908, -173.265]
  Call Extruder(1183.713)
  MoveL 1912 to (41.12, 52.43, 12.6) mm, rotated rx 0 ry 90 rz 0 deg; joints [-10.184, 2.502, 54.947, 167.969, 58.023, -173.56]
  Call Extruder(1184.925)
  MoveL 1913 to (47.56, 58.88, 12.6) mm, rotated rx 0 ry 90 rz 0 deg; joints [-10.516, 3.102, 53.264, 167.431, 57.005, -173.077]
  Call Extruder(1185.573)
  MoveL 1914 to (52.43, 58.88, 12.6) mm, rotated rx 0 ry 90 rz 0 deg; joints [-10.46, 3.502, 52.16, 167.397, 56.31, -172.93]
  Call Extruder(1186.611)
  MoveL 1915 to (57.95, 53.36, 12.6) mm, rotated rx 0 ry 90 rz 0 deg; joints [-10.054, 3.885, 51.112, 167.786, 55.611, -173.03]
  Call Extruder(1186.735)
  MoveL 1916 to (58.88, 53.37, 12.6) mm, rotated rx 0 ry 90 rz 0 deg; joints [-10.044, 3.965, 50.893, 167.778, 55.474, -173.001]
  Call Extruder(1187.469)
  MoveL 1917 to (58.88, 58.88, 12.6) mm, rotated rx 0 ry 90 rz 0 deg; joints [-10.386, 4.052, 50.658, 167.344, 55.372, -172.728]
  Call Extruder(1187.469)
  MoveL 1918 to (58.88, 58.88, 12.6) mm, rotated rx 0 ry 90 rz 0 deg; joints [-10.386, 4.052, 50.658, 167.344, 55.372, -172.728]
  Call Extruder(1190.810)
  MoveL 1919 to (41.12, 41.12, 12.6) mm, rotated rx 0 ry 90 rz 0 deg; joints [-9.467, 2.352, 55.371, 168.843, 58.215, -174.069]
  Call Extruder(1191.668)
  MoveL 1920 to (41.12, 47.56, 12.6) mm, rotated rx 0 ry 90 rz 0 deg; joints [-9.876, 2.436, 55.134, 168.345, 58.107, -173.781]
  Call Extruder(1192.615)
  MoveL 1921 to (46.15, 42.53, 12.6) mm, rotated rx 0 ry 90 rz 0 deg; joints [-9.503, 2.76, 54.221, 168.71, 57.49, -173.876]
  Call Extruder(1192.679)
  MoveL 1922 to (46.15, 43.02, 12.6) mm, rotated rx 0 ry 90 rz 0 deg; joints [-9.534, 2.766, 54.203, 168.672, 57.482, -173.854]
  Call Extruder(1193.209)
  MoveL 1923 to (50.13, 43.02, 12.6) mm, rotated rx 0 ry 90 rz 0 deg; joints [-9.492, 3.084, 53.316, 168.65, 56.92, -173.747]
  Call Extruder(1193.583)
  MoveL 1924 to (52.95, 43.02, 12.6) mm, rotated rx 0 ry 90 rz 0 deg; joints [-9.462, 3.314, 52.679, 168.632, 56.517, -173.671]
  Call Extruder(1193.836)
  MoveL 1925 to (52.95, 41.12, 12.6) mm, rotated rx 0 ry 90 rz 0 deg; joints [-9.343, 3.288, 52.751, 168.78, 56.549, -173.76]
  Call Extruder(1194.625)
  MoveL 1926 to (58.88, 41.12, 12.6) mm, rotated rx 0 ry 90 rz 0 deg; joints [-9.282, 3.786, 51.383, 168.739, 55.689, -173.596]
  MoveL 1927 to (59.08, 41.12, 12.6) mm, rotated rx 0 ry 90 rz 0 deg; joints [-9.28, 3.803, 51.336, 168.737, 55.659, -173.59]
  Set speed (120.0 mm/s)
  MoveL 1928 to (52.3, 42.37, 12.6) mm, rotated rx 0 ry 90 rz 0 deg; joints [-9.428, 3.251, 52.851, 168.687, 56.621, -173.719]
  Set speed (1000.0 mm/s)
  MoveL 1929 to (52.23, 42.3, 12.6) mm, rotated rx 0 ry 90 rz 0 deg; joints [-9.425, 3.245, 52.87, 168.693, 56.632, -173.724]
  Set speed (30.0 mm/s)
  Call Extruder(1194.679)
  MoveL 1930 to (52.23, 41.9, 12.6) mm, rotated rx 0 ry 90 rz 0 deg; joints [-9.4, 3.239, 52.885, 168.724, 56.639, -173.743]
  Call Extruder(1194.825)
  MoveL 1931 to (52.23, 40.8, 12.6) mm, rotated rx 0 ry 90 rz 0 deg; joints [-9.33, 3.224, 52.926, 168.809, 56.658, -173.794]
  Call Extruder(1194.878)
  MoveL 1932 to (52.23, 40.4, 12.6) mm, rotated rx 0 ry 90 rz 0 deg; joints [-9.305, 3.219, 52.941, 168.841, 56.664, -173.813]
  Call Extruder(1194.913)
  MoveL 1933 to (52.63, 40.4, 12.6) mm, rotated rx 0 ry 90 rz 0 deg; joints [-9.301, 3.252, 52.85, 168.838, 56.607, -173.802]
  Call Extruder(1195.840)
  MoveL 1934 to (59.6, 40.4, 12.6) mm, rotated rx 0 ry 90 rz 0 deg; joints [-9.23, 3.837, 51.241, 168.79, 55.595, -173.61]
  Call Extruder(1196.647)
  MoveL 1935 to (59.6, 46.46, 12.6) mm, rotated rx 0 ry 90 rz 0 deg; joints [-9.608, 3.924, 51.005, 168.315, 55.491, -173.317]
  Call Extruder(1196.904)
  MoveL 1936 to (57.67, 46.47, 12.6) mm, rotated rx 0 ry 90 rz 0 deg; joints [-9.628, 3.758, 51.457, 168.33, 55.774, -173.373]
  Call Extruder(1197.182)
  MoveL 1937 to (57.67, 48.56, 12.6) mm, rotated rx 0 ry 90 rz 0 deg; joints [-9.759, 3.789, 51.374, 168.166, 55.738, -173.272]
  Call Extruder(1197.235)
  MoveL 1938 to (57.67, 48.96, 12.6) mm, rotated rx 0 ry 90 rz 0 deg; joints [-9.783, 3.795, 51.358, 168.134, 55.731, -173.253]
  Call Extruder(1197.270)
  MoveL 1939 to (58.07, 48.96, 12.6) mm, rotated rx 0 ry 90 rz 0 deg; joints [-9.779, 3.829, 51.264, 168.131, 55.672, -173.241]
  Call Extruder(1197.474)
  MoveL 1940 to (59.6, 48.96, 12.6) mm, rotated rx 0 ry 90 rz 0 deg; joints [-9.763, 3.961, 50.904, 168.119, 55.447, -173.195]
  Call Extruder(1197.634)
  MoveL 1941 to (59.6, 50.16, 12.6) mm, rotated rx 0 ry 90 rz 0 deg; joints [-9.838, 3.979, 50.855, 168.024, 55.426, -173.136]
  Call Extruder(1197.838)
  MoveL 1942 to (58.07, 50.16, 12.6) mm, rotated rx 0 ry 90 rz 0 deg; joints [-9.854, 3.847, 51.216, 168.037, 55.651, -173.182]
  Call Extruder(1197.891)
  MoveL 1943 to (57.67, 50.16, 12.6) mm, rotated rx 0 ry 90 rz 0 deg; joints [-9.858, 3.812, 51.31, 168.04, 55.71, -173.194]
  Call Extruder(1197.926)
  MoveL 1944 to (57.67, 50.56, 12.6) mm, rotated rx 0 ry 90 rz 0 deg; joints [-9.883, 3.818, 51.293, 168.009, 55.703, -173.175]
  Call Extruder(1198.203)
  MoveL 1945 to (57.67, 52.64, 12.6) mm, rotated rx 0 ry 90 rz 0 deg; joints [-10.013, 3.85, 51.208, 167.845, 55.665, -173.074]
  Call Extruder(1198.460)
  MoveL 1946 to (59.6, 52.65, 12.6) mm, rotated rx 0 ry 90 rz 0 deg; joints [-9.992, 4.017, 50.753, 167.829, 55.381, -173.014]
  Call Extruder(1199.385)
  MoveL 1947 to (59.6, 59.6, 12.6) mm, rotated rx 0 ry 90 rz 0 deg; joints [-10.423, 4.127, 50.456, 167.281, 55.252, -172.669]
  Call Extruder(1201.939)
  MoveL 1948 to (40.4, 59.6, 12.6) mm, rotated rx 0 ry 90 rz 0 deg; joints [-10.646, 2.548, 54.817, 167.417, 57.994, -173.253]
  Call Extruder(1204.494)
  MoveL 1949 to (40.4, 40.4, 12.6) mm, rotated rx 0 ry 90 rz 0 deg; joints [-9.429, 2.288, 55.552, 168.902, 58.326, -174.119]
  Call Extruder(1205.302)
  MoveL 1950 to (46.47, 40.4, 12.6) mm, rotated rx 0 ry 90 rz 0 deg; joints [-9.365, 2.757, 54.228, 168.873, 57.48, -173.964]
  Call Extruder(1205.355)
  MoveL 1951 to (46.87, 40.4, 12.6) mm, rotated rx 0 ry 90 rz 0 deg; joints [-9.361, 2.789, 54.14, 168.871, 57.424, -173.954]
  Call Extruder(1205.389)
  MoveL 1952 to (46.87, 40.8, 12.6) mm, rotated rx 0 ry 90 rz 0 deg; joints [-9.386, 2.794, 54.125, 168.84, 57.417, -173.936]
  Call Extruder(1205.536)
  MoveL 1953 to (46.87, 41.9, 12.6) mm, rotated rx 0 ry 90 rz 0 deg; joints [-9.456, 2.808, 54.085, 168.755, 57.399, -173.886]
  Call Extruder(1205.589)
  MoveL 1954 to (46.87, 42.3, 12.6) mm, rotated rx 0 ry 90 rz 0 deg; joints [-9.481, 2.814, 54.07, 168.724, 57.393, -173.867]
  Call Extruder(1205.623)
  MoveL 1955 to (47.27, 42.3, 12.6) mm, rotated rx 0 ry 90 rz 0 deg; joints [-9.477, 2.845, 53.982, 168.722, 57.337, -173.857]
  Call Extruder(1205.897)
  MoveL 1956 to (49.33, 42.3, 12.6) mm, rotated rx 0 ry 90 rz 0 deg; joints [-9.455, 3.01, 53.523, 168.71, 57.045, -173.802]
  Call Extruder(1206.150)
  MoveL 1957 to (49.33, 40.4, 12.6) mm, rotated rx 0 ry 90 rz 0 deg; joints [-9.335, 2.985, 53.593, 168.858, 57.077, -173.89]
  Call Extruder(1206.213)
  MoveL 1958 to (49.81, 40.4, 12.6) mm, rotated rx 0 ry 90 rz 0 deg; joints [-9.33, 3.023, 53.487, 168.855, 57.009, -173.877]
  Call Extruder(1206.363)
  MoveL 1959 to (49.81, 42.3, 12.6) mm, rotated rx 0 ry 90 rz 0 deg; joints [-9.45, 3.048, 53.416, 168.707, 56.978, -173.789]
  Call Extruder(1206.632)
  MoveL 1960 to (51.83, 42.3, 12.6) mm, rotated rx 0 ry 90 rz 0 deg; joints [-9.429, 3.212, 52.961, 168.695, 56.69, -173.735]
  Call Extruder(1206.666)
  MoveL 1961 to (52.23, 42.3, 12.6) mm, rotated rx 0 ry 90 rz 0 deg; joints [-9.425, 3.245, 52.87, 168.693, 56.632, -173.724]
  Set speed (120.0 mm/s)
  MoveL 1962 to (52.23, 41.9, 12.6) mm, rotated rx 0 ry 90 rz 0 deg; joints [-9.4, 3.239, 52.885, 168.724, 56.639, -173.743]
  Set speed (1000.0 mm/s)
  MoveL 1963 to (52.33, 41.9, 12.6) mm, rotated rx 0 ry 90 rz 0 deg; joints [-9.398, 3.247, 52.862, 168.723, 56.625, -173.74]
  MoveL 1964 to (57.25, 49.33, 12.6) mm, rotated rx 0 ry 90 rz 0 deg; joints [-9.811, 3.765, 51.44, 168.108, 55.785, -173.247]
  MoveL 1965 to (57.48, 49.56, 12.6) mm, rotated rx 0 ry 90 rz 0 deg; joints [-9.823, 3.787, 51.378, 168.089, 55.748, -173.229]
  Set speed (30.0 mm/s)
  Call Extruder(1206.725)
  MoveL 1966 to (58.04, 49.56, 12.6) mm, rotated rx 0 ry 90 rz 0 deg; joints [-9.817, 3.836, 51.246, 168.084, 55.665, -173.212]
  Call Extruder(1206.832)
